LIN {X 0,Y 305.459,Z 160.438,A -85,B 0,C 180,E1 -15804.888,E2 -15804.888} C_VEL
LIN {X 0,Y 305.449,Z 160.435,A -85,B 0,C 180,E1 -15808.356,E2 -15808.356} C_VEL
LIN {X 0,Y 305.518,Z 160.428,A -85,B 0,C 180,E1 -15811.115,E2 -15811.115} C_VEL
LIN {X 0,Y 305.57,Z 160.425,A -85,B 0,C 180,E1 -15814.089,E2 -15814.089} C_VEL
LIN {X 0,Y 305.497,Z 160.431,A -85,B 0,C 180,E1 -15818.404,E2 -15818.404} C_VEL
LIN {X 0,Y 305.556,Z 160.425,A -85,B 0,C 180,E1 -15821.217,E2 -15821.217} C_VEL
LIN {X 0,Y 305.626,Z 160.413,A -85,B 0,C 180,E1 -15825.349,E2 -15825.349} C_VEL
LIN {X 0,Y 305.625,Z 160.413,A -85,B 0,C 180,E1 -15829.4,E2 -15829.4} C_VEL
LIN {X 0,Y 305.749,Z 160.391,A -85,B 0,C 180,E1 -15832.074,E2 -15832.074} C_VEL
LIN {X 0,Y 305.671,Z 160.401,A -85,B 0,C 180,E1 -15834.724,E2 -15834.724} C_VEL
LIN {X 0,Y 305.952,Z 160.37,A -85,B 0,C 180,E1 -15838.685,E2 -15838.685} C_VEL
LIN {X 0,Y 305.948,Z 160.361,A -85,B 0,C 180,E1 -15841.317,E2 -15841.317} C_VEL
LIN {X 0,Y 305.789,Z 160.382,A -85,B 0,C 180,E1 -15846.6,E2 -15846.6} C_VEL
LIN {X 0,Y 305.696,Z 160.401,A -85,B 0,C 180,E1 -15849.262,E2 -15849.262} C_VEL
LIN {X 0,Y 305.587,Z 160.417,A -85,B 0,C 180,E1 -15853.297,E2 -15853.297} C_VEL
LIN {X 0,Y 305.541,Z 160.413,A -85,B 0,C 180,E1 -15856.024,E2 -15856.024} C_VEL
LIN {X 0,Y 305.482,Z 160.427,A -85,B 0,C 180,E1 -15860.189,E2 -15860.189} C_VEL
LIN {X 0,Y 305.442,Z 160.436,A -85,B 0,C 180,E1 -15864.468,E2 -15864.468} C_VEL
LIN {X 0,Y 305.451,Z 160.431,A -85,B 0,C 180,E1 -15867.399,E2 -15867.399} C_VEL
LIN {X 0,Y 305.431,Z 160.429,A -85,B 0,C 180,E1 -15870.414,E2 -15870.414} C_VEL
LIN {X 0,Y 305.467,Z 160.428,A -85,B 0,C 180,E1 -15874.079,E2 -15874.079} C_VEL
LIN {X 0,Y 305.453,Z 160.438,A -85,B 0,C 180,E1 -15876.744,E2 -15876.744} C_VEL
LIN {X 0,Y 305.411,Z 160.442,A -85,B 0,C 180,E1 -15880.59,E2 -15880.59} C_VEL
LIN {X 0,Y 305.423,Z 160.441,A -85,B 0,C 180,E1 -15883.657,E2 -15883.657} C_VEL
LIN {X 0,Y 305.437,Z 160.444,A -85,B 0,C 180,E1 -15887.419,E2 -15887.419} C_VEL
LIN {X 0,Y 305.444,Z 160.439,A -85,B 0,C 180,E1 -15891.593,E2 -15891.593} C_VEL
LIN {X 0,Y 305.489,Z 160.556,A -85,B 0,C 180,E1 -15895.319,E2 -15895.319} C_VEL
LIN {X 0,Y 308.003,Z 170.762,A -85,B 0,C 180,E1 -15898.728,E2 -15898.728} C_VEL
LIN {X 0,Y 309.903,Z 179.796,A -85,B 0,C 180,E1 -15901.56,E2 -15901.56} C_VEL
LIN {X 0,Y 310.831,Z 184.661,A -85,B 0,C 180,E1 -15902.985,E2 -15902.985} C_VEL
LIN {X 0,Y 312.383,Z 189.96,A -85,B 0,C 180,E1 -15903.288,E2 -15903.288} C_VEL
LIN {X 0,Y 316.289,Z 210.278,A -85,B 0,C 180,E1 -15904.21,E2 -15904.21} C_VEL
LIN {X 0,Y 318.973,Z 229.13,A -85,B 0,C 180,E1 -15904.953,E2 -15904.953} C_VEL
LIN {X 0,Y 317.191,Z 294.073,A -85,B 0,C 180,E1 -15906.495,E2 -15906.495} C_VEL
LIN {X 0,Y 316.159,Z 307.688,A -85,B 0,C 180,E1 -15907.064,E2 -15907.064} C_VEL
LIN {X 0,Y 314.832,Z 320.533,A -85,B 0,C 180,E1 -15907.871,E2 -15907.871} C_VEL
LIN {X 0,Y 313.273,Z 333.066,A -85,B 0,C 180,E1 -15908.965,E2 -15908.965} C_VEL
LIN {X 0,Y 311.564,Z 344.273,A -85,B 0,C 180,E1 -15910.223,E2 -15910.223} C_VEL
LIN {X 0,Y 309.857,Z 354.387,A -85,B 0,C 180,E1 -15911.657,E2 -15911.657} C_VEL
LIN {X 0,Y 308.403,Z 363.848,A -85,B 0,C 180,E1 -15913.345,E2 -15913.345} C_VEL
LIN {X 0,Y 307.067,Z 371.791,A -85,B 0,C 180,E1 -15915.079,E2 -15915.079} C_VEL
LIN {X 0,Y 305.664,Z 379.121,A -85,B 0,C 180,E1 -15917.046,E2 -15917.046} C_VEL
LIN {X 0,Y 304.863,Z 384.095,A -85,B 0,C 180,E1 -15918.7,E2 -15918.7} C_VEL
LIN {X 0,Y 304.229,Z 388.944,A -85,B 0,C 180,E1 -15920.694,E2 -15920.694} C_VEL
LIN {X 0,Y 303.828,Z 392.677,A -85,B 0,C 180,E1 -15922.691,E2 -15922.691} C_VEL
LIN {X 0,Y 303.621,Z 395.397,A -85,B 0,C 180,E1 -15924.688,E2 -15924.688} C_VEL
LIN {X 0,Y 303.629,Z 396.691,A -85,B 0,C 180,E1 -15926.018,E2 -15926.018} C_VEL
LIN {X 0,Y 303.624,Z 397.581,A -85,B 0,C 180,E1 -15927.347,E2 -15927.347} C_VEL
LIN {X 0,Y 303.615,Z 398.031,A -85,B 0,C 180,E1 -15928.674,E2 -15928.674} C_VEL
LIN {X 0,Y 303.67,Z 398.088,A -85,B 0,C 180,E1 -15930,E2 -15930} C_VEL
LIN {X 0,Y 303.626,Z 397.751,A -85,B 0,C 180,E1 -15931.327,E2 -15931.327} C_VEL
LIN {X 0,Y 303.626,Z 397.019,A -85,B 0,C 180,E1 -15932.654,E2 -15932.654} C_VEL
LIN {X 0,Y 303.63,Z 395.835,A -85,B 0,C 180,E1 -15933.982,E2 -15933.982} C_VEL
LIN {X 0,Y 303.622,Z 393.936,A -85,B 0,C 180,E1 -15935.532,E2 -15935.532} C_VEL
LIN {X 0,Y 303.927,Z 389.712,A -85,B 0,C 180,E1 -15937.975,E2 -15937.975} C_VEL
LIN {X 0,Y 304.361,Z 385.011,A -85,B 0,C 180,E1 -15939.973,E2 -15939.973} C_VEL
LIN {X 0,Y 305.191,Z 377.914,A -85,B 0,C 180,E1 -15942.299,E2 -15942.299} C_VEL
LIN {X 0,Y 306.358,Z 370.227,A -85,B 0,C 180,E1 -15944.277,E2 -15944.277} C_VEL
LIN {X 0,Y 307.697,Z 360.747,A -85,B 0,C 180,E1 -15946.21,E2 -15946.21} C_VEL
LIN {X 0,Y 309.019,Z 350.537,A -85,B 0,C 180,E1 -15947.881,E2 -15947.881} C_VEL
LIN {X 0,Y 310.561,Z 339.27,A -85,B 0,C 180,E1 -15949.328,E2 -15949.328} C_VEL
LIN {X 0,Y 311.897,Z 328.23,A -85,B 0,C 180,E1 -15950.443,E2 -15950.443} C_VEL
LIN {X 0,Y 313.162,Z 316.02,A -85,B 0,C 180,E1 -15951.389,E2 -15951.389} C_VEL
LIN {X 0,Y 314.23,Z 303.288,A -85,B 0,C 180,E1 -15952.088,E2 -15952.088} C_VEL
LIN {X 0,Y 314.859,Z 290.01,A -85,B 0,C 180,E1 -15952.558,E2 -15952.558} C_VEL
LIN {X 0,Y 316.214,Z 227.211,A -85,B 0,C 180,E1 -15954.02,E2 -15954.02} C_VEL
LIN {X 0,Y 310.529,Z 189.601,A -85,B 0,C 180,E1 -15955.391,E2 -15955.391} C_VEL
LIN {X 0,Y 309.869,Z 185.486,A -85,B 0,C 180,E1 -15955.572,E2 -15955.572} C_VEL
LIN {X 0,Y 309.869,Z 181.695,A -85,B 0,C 180,E1 -15956.612,E2 -15956.612} C_VEL
LIN {X 0,Y 307.783,Z 170.867,A -85,B 0,C 180,E1 -15959.806,E2 -15959.806} C_VEL
LIN {X 0,Y 305.485,Z 160.432,A -85,B 0,C 180,E1 -15963.071,E2 -15963.071} C_VEL
LIN {X 0,Y 305.457,Z 160.435,A -85,B 0,C 180,E1 -15966.743,E2 -15966.743} C_VEL
LIN {X 0,Y 305.414,Z 160.44,A -85,B 0,C 180,E1 -15970.59,E2 -15970.59} C_VEL
LIN {X 0,Y 305.425,Z 160.44,A -85,B 0,C 180,E1 -15973.656,E2 -15973.656} C_VEL
LIN {X 0,Y 305.44,Z 160.44,A -85,B 0,C 180,E1 -15977.418,E2 -15977.418} C_VEL
LIN {X 0,Y 305.465,Z 160.435,A -85,B 0,C 180,E1 -15981.595,E2 -15981.595} C_VEL
LIN {X 0,Y 305.466,Z 160.437,A -85,B 0,C 180,E1 -15984.886,E2 -15984.886} C_VEL
LIN {X 0,Y 305.447,Z 160.436,A -85,B 0,C 180,E1 -15988.358,E2 -15988.358} C_VEL
LIN {X 0,Y 305.48,Z 160.434,A -85,B 0,C 180,E1 -15991.109,E2 -15991.109} C_VEL
LIN {X 0,Y 305.505,Z 160.428,A -85,B 0,C 180,E1 -15994.081,E2 -15994.081} C_VEL
LIN {X 0,Y 305.478,Z 160.434,A -85,B 0,C 180,E1 -15996.975,E2 -15996.975} C_VEL
LIN {X 0,Y 305.513,Z 160.427,A -85,B 0,C 180,E1 -16001.212,E2 -16001.212} C_VEL
LIN {X 0,Y 305.584,Z 160.418,A -85,B 0,C 180,E1 -16005.345,E2 -16005.345} C_VEL
LIN {X 0,Y 305.628,Z 160.41,A -85,B 0,C 180,E1 -16009.398,E2 -16009.398} C_VEL
LIN {X 0,Y 305.751,Z 160.393,A -85,B 0,C 180,E1 -16012.072,E2 -16012.072} C_VEL
LIN {X 0,Y 305.662,Z 160.409,A -85,B 0,C 180,E1 -16014.722,E2 -16014.722} C_VEL
LIN {X 0,Y 305.939,Z 160.374,A -85,B 0,C 180,E1 -16018.683,E2 -16018.683} C_VEL
LIN {X 0,Y 305.939,Z 160.37,A -85,B 0,C 180,E1 -16021.315,E2 -16021.315} C_VEL
LIN {X 0,Y 305.787,Z 160.392,A -85,B 0,C 180,E1 -16026.598,E2 -16026.598} C_VEL
LIN {X 0,Y 305.696,Z 160.404,A -85,B 0,C 180,E1 -16029.26,E2 -16029.26} C_VEL
LIN {X 0,Y 305.572,Z 160.417,A -85,B 0,C 180,E1 -16033.296,E2 -16033.296} C_VEL
LIN {X 0,Y 305.512,Z 160.423,A -85,B 0,C 180,E1 -16036.023,E2 -16036.023} C_VEL
LIN {X 0,Y 305.476,Z 160.432,A -85,B 0,C 180,E1 -16040.187,E2 -16040.187} C_VEL
LIN {X 0,Y 305.439,Z 160.433,A -85,B 0,C 180,E1 -16044.466,E2 -16044.466} C_VEL
LIN {X 0,Y 305.441,Z 160.432,A -85,B 0,C 180,E1 -16047.398,E2 -16047.398} C_VEL
LIN {X 0,Y 305.416,Z 160.437,A -85,B 0,C 180,E1 -16050.413,E2 -16050.413} C_VEL
LIN {X 0,Y 305.463,Z 160.433,A -85,B 0,C 180,E1 -16054.077,E2 -16054.077} C_VEL
LIN {X 0,Y 305.45,Z 160.432,A -85,B 0,C 180,E1 -16056.741,E2 -16056.741} C_VEL
LIN {X 0,Y 305.406,Z 160.438,A -85,B 0,C 180,E1 -16060.588,E2 -16060.588} C_VEL
LIN {X 0,Y 305.417,Z 160.44,A -85,B 0,C 180,E1 -16063.655,E2 -16063.655} C_VEL
LIN {X 0,Y 305.431,Z 160.436,A -85,B 0,C 180,E1 -16067.417,E2 -16067.417} C_VEL
LIN {X 0,Y 305.455,Z 160.435,A -85,B 0,C 180,E1 -16071.594,E2 -16071.594} C_VEL
LIN {X 0,Y 305.456,Z 160.435,A -85,B 0,C 180,E1 -16074.885,E2 -16074.885} C_VEL
LIN {X 0,Y 305.436,Z 160.438,A -85,B 0,C 180,E1 -16078.357,E2 -16078.357} C_VEL
LIN {X 0,Y 305.468,Z 160.432,A -85,B 0,C 180,E1 -16081.108,E2 -16081.108} C_VEL
LIN {X 0,Y 305.472,Z 160.432,A -85,B 0,C 180,E1 -16084.078,E2 -16084.078} C_VEL
LIN {X 0,Y 305.452,Z 160.436,A -85,B 0,C 180,E1 -16088.399,E2 -16088.399} C_VEL
LIN {X 0,Y 305.502,Z 160.429,A -85,B 0,C 180,E1 -16091.212,E2 -16091.212} C_VEL
LIN {X 0,Y 305.572,Z 160.418,A -85,B 0,C 180,E1 -16095.345,E2 -16095.345} C_VEL
LIN {X 0,Y 305.615,Z 160.413,A -85,B 0,C 180,E1 -16099.399,E2 -16099.399} C_VEL
LIN {X 0,Y 305.739,Z 160.401,A -85,B 0,C 180,E1 -16102.072,E2 -16102.072} C_VEL
LIN {X 0,Y 305.65,Z 160.457,A -85,B 0,C 180,E1 -16104.722,E2 -16104.722} C_VEL
LIN {X 0,Y 306.613,Z 165.016,A -85,B 0,C 180,E1 -16106.248,E2 -16106.248} C_VEL
LIN {X 0,Y 312.464,Z 179.943,A -85,B 0,C 180,E1 -16107.106,E2 -16107.106} C_VEL
LIN {X 0,Y 315.894,Z 190.278,A -85,B 0,C 180,E1 -16107.63,E2 -16107.63} C_VEL
LIN {X 0,Y 316.999,Z 196.484,A -85,B 0,C 180,E1 -16107.866,E2 -16107.866} C_VEL
LIN {X 0,Y 314.976,Z 272.651,A -85,B 0,C 180,E1 -16109.64,E2 -16109.64} C_VEL
LIN {X 0,Y 314.278,Z 285.795,A -85,B 0,C 180,E1 -16110.2,E2 -16110.2} C_VEL
LIN {X 0,Y 313.454,Z 297.884,A -85,B 0,C 180,E1 -16110.963,E2 -16110.963} C_VEL
LIN {X 0,Y 312.447,Z 309.33,A -85,B 0,C 180,E1 -16111.933,E2 -16111.933} C_VEL
LIN {X 0,Y 311.048,Z 321.197,A -85,B 0,C 180,E1 -16113.238,E2 -16113.238} C_VEL
LIN {X 0,Y 309.738,Z 331.319,A -85,B 0,C 180,E1 -16114.641,E2 -16114.641} C_VEL
LIN {X 0,Y 308.483,Z 340.503,A -85,B 0,C 180,E1 -16116.212,E2 -16116.212} C_VEL
LIN {X 0,Y 307.288,Z 348.479,A -85,B 0,C 180,E1 -16117.887,E2 -16117.887} C_VEL
LIN {X 0,Y 306.119,Z 356.027,A -85,B 0,C 180,E1 -16119.848,E2 -16119.848} C_VEL
LIN {X 0,Y 305.158,Z 362.491,A -85,B 0,C 180,E1 -16121.963,E2 -16121.963} C_VEL
LIN {X 0,Y 304.444,Z 367.731,A -85,B 0,C 180,E1 -16124.179,E2 -16124.179} C_VEL
LIN {X 0,Y 304.015,Z 371.135,A -85,B 0,C 180,E1 -16126.105,E2 -16126.105} C_VEL
LIN {X 0,Y 303.636,Z 373.968,A -85,B 0,C 180,E1 -16128.383,E2 -16128.383} C_VEL
LIN {X 0,Y 303.447,Z 375.408,A -85,B 0,C 180,E1 -16130.329,E2 -16130.329} C_VEL
LIN {X 0,Y 303.451,Z 375.955,A -85,B 0,C 180,E1 -16132.122,E2 -16132.122} C_VEL
LIN {X 0,Y 303.575,Z 375.564,A -85,B 0,C 180,E1 -16134.627,E2 -16134.627} C_VEL
LIN {X 0,Y 303.751,Z 374.658,A -85,B 0,C 180,E1 -16136.079,E2 -16136.079} C_VEL
LIN {X 0,Y 304.286,Z 371.901,A -85,B 0,C 180,E1 -16138.64,E2 -16138.64} C_VEL
LIN {X 0,Y 304.946,Z 367.905,A -85,B 0,C 180,E1 -16141.021,E2 -16141.021} C_VEL
LIN {X 0,Y 305.631,Z 364.099,A -85,B 0,C 180,E1 -16142.71,E2 -16142.71} C_VEL
LIN {X 0,Y 306.836,Z 357.731,A -85,B 0,C 180,E1 -16144.933,E2 -16144.933} C_VEL
LIN {X 0,Y 308.34,Z 349.761,A -85,B 0,C 180,E1 -16147.086,E2 -16147.086} C_VEL
LIN {X 0,Y 309.942,Z 340.851,A -85,B 0,C 180,E1 -16148.994,E2 -16148.994} C_VEL
LIN {X 0,Y 311.578,Z 331.082,A -85,B 0,C 180,E1 -16150.653,E2 -16150.653} C_VEL
LIN {X 0,Y 313.215,Z 320.303,A -85,B 0,C 180,E1 -16152.118,E2 -16152.118} C_VEL
LIN {X 0,Y 314.771,Z 308.639,A -85,B 0,C 180,E1 -16153.359,E2 -16153.359} C_VEL
LIN {X 0,Y 315.985,Z 296.732,A -85,B 0,C 180,E1 -16154.333,E2 -16154.333} C_VEL
LIN {X 0,Y 316.947,Z 284.09,A -85,B 0,C 180,E1 -16155.093,E2 -16155.093} C_VEL
LIN {X 0,Y 317.614,Z 271.593,A -85,B 0,C 180,E1 -16155.586,E2 -16155.586} C_VEL
LIN {X 0,Y 319.739,Z 196.647,A -85,B 0,C 180,E1 -16157.338,E2 -16157.338} C_VEL
LIN {X 0,Y 318.932,Z 193.583,A -85,B 0,C 180,E1 -16157.495,E2 -16157.495} C_VEL
LIN {X 0,Y 316.079,Z 188.881,A -85,B 0,C 180,E1 -16157.897,E2 -16157.897} C_VEL
LIN {X 0,Y 304.505,Z 175.175,A -85,B 0,C 180,E1 -16159.481,E2 -16159.481} C_VEL
LIN {X 0,Y 301.74,Z 170.475,A -85,B 0,C 180,E1 -16159.924,E2 -16159.924} C_VEL
LIN {X 0,Y 299.63,Z 166.062,A -85,B 0,C 180,E1 -16160.327,E2 -16160.327} C_VEL
LIN {X 0,Y 298.456,Z 161.318,A -85,B 0,C 180,E1 -16162.152,E2 -16162.152} C_VEL
LIN {X 0,Y 298.405,Z 161.318,A -85,B 0,C 180,E1 -16165.582,E2 -16165.582} C_VEL
LIN {X 0,Y 298.392,Z 161.315,A -85,B 0,C 180,E1 -16168.792,E2 -16168.792} C_VEL
LIN {X 0,Y 298.461,Z 161.309,A -85,B 0,C 180,E1 -16171.906,E2 -16171.906} C_VEL
LIN {X 0,Y 298.484,Z 161.307,A -85,B 0,C 180,E1 -16174.925,E2 -16174.925} C_VEL
LIN {X 0,Y 298.444,Z 161.306,A -85,B 0,C 180,E1 -16179.316,E2 -16179.316} C_VEL
LIN {X 0,Y 298.508,Z 161.298,A -85,B 0,C 180,E1 -16182.179,E2 -16182.179} C_VEL
LIN {X 0,Y 298.585,Z 161.293,A -85,B 0,C 180,E1 -16184.996,E2 -16184.996} C_VEL
LIN {X 0,Y 298.583,Z 161.292,A -85,B 0,C 180,E1 -16189.147,E2 -16189.147} C_VEL
LIN {X 0,Y 298.7,Z 161.269,A -85,B 0,C 180,E1 -16191.886,E2 -16191.886} C_VEL
LIN {X 0,Y 298.639,Z 161.278,A -85,B 0,C 180,E1 -16194.6,E2 -16194.6} C_VEL
LIN {X 0,Y 298.919,Z 161.246,A -85,B 0,C 180,E1 -16198.654,E2 -16198.654} C_VEL
LIN {X 0,Y 298.915,Z 161.236,A -85,B 0,C 180,E1 -16201.348,E2 -16201.348} C_VEL
LIN {X 0,Y 298.737,Z 161.261,A -85,B 0,C 180,E1 -16206.756,E2 -16206.756} C_VEL
LIN {X 0,Y 298.628,Z 161.283,A -85,B 0,C 180,E1 -16209.483,E2 -16209.483} C_VEL
LIN {X 0,Y 298.543,Z 161.297,A -85,B 0,C 180,E1 -16213.617,E2 -16213.617} C_VEL
LIN {X 0,Y 298.473,Z 161.293,A -85,B 0,C 180,E1 -16216.414,E2 -16216.414} C_VEL
LIN {X 0,Y 298.441,Z 161.31,A -85,B 0,C 180,E1 -16219.616,E2 -16219.616} C_VEL
LIN {X 0,Y 298.384,Z 161.317,A -85,B 0,C 180,E1 -16223.605,E2 -16223.605} C_VEL
LIN {X 0,Y 298.404,Z 161.304,A -85,B 0,C 180,E1 -16226.584,E2 -16226.584} C_VEL
LIN {X 0,Y 298.395,Z 161.309,A -85,B 0,C 180,E1 -16229.645,E2 -16229.645} C_VEL
LIN {X 0,Y 298.395,Z 161.316,A -85,B 0,C 180,E1 -16232.801,E2 -16232.801} C_VEL
LIN {X 0,Y 298.428,Z 161.313,A -85,B 0,C 180,E1 -16236.803,E2 -16236.803} C_VEL
LIN {X 0,Y 298.349,Z 161.32,A -85,B 0,C 180,E1 -16241.269,E2 -16241.269} C_VEL
LIN {X 0,Y 298.357,Z 161.326,A -85,B 0,C 180,E1 -16245.036,E2 -16245.036} C_VEL
LIN {X 0,Y 298.35,Z 161.324,A -85,B 0,C 180,E1 -16248.922,E2 -16248.922} C_VEL
LIN {X 0,Y 298.429,Z 161.303,A -85,B 0,C 180,E1 -16253.198,E2 -16253.198} C_VEL
LIN {X 0,Y 298.463,Z 161.48,A -85,B 0,C 180,E1 -16254.662,E2 -16254.662} C_VEL
LIN {X 0,Y 301.06,Z 172.051,A -85,B 0,C 180,E1 -16258.315,E2 -16258.315} C_VEL
LIN {X 0,Y 303.12,Z 181.821,A -85,B 0,C 180,E1 -16261.46,E2 -16261.46} C_VEL
LIN {X 0,Y 303.597,Z 184.363,A -85,B 0,C 180,E1 -16262.2,E2 -16262.2} C_VEL
LIN {X 0,Y 306.198,Z 191.246,A -85,B 0,C 180,E1 -16262.674,E2 -16262.674} C_VEL
LIN {X 0,Y 309.548,Z 208.929,A -85,B 0,C 180,E1 -16263.508,E2 -16263.508} C_VEL
LIN {X 0,Y 312.601,Z 228.987,A -85,B 0,C 180,E1 -16264.345,E2 -16264.345} C_VEL
LIN {X 0,Y 310.814,Z 293.869,A -85,B 0,C 180,E1 -16265.925,E2 -16265.925} C_VEL
LIN {X 0,Y 309.741,Z 307.694,A -85,B 0,C 180,E1 -16266.516,E2 -16266.516} C_VEL
LIN {X 0,Y 308.434,Z 319.935,A -85,B 0,C 180,E1 -16267.298,E2 -16267.298} C_VEL
LIN {X 0,Y 306.894,Z 331.737,A -85,B 0,C 180,E1 -16268.33,E2 -16268.33} C_VEL
LIN {X 0,Y 305.11,Z 343.124,A -85,B 0,C 180,E1 -16269.611,E2 -16269.611} C_VEL
LIN {X 0,Y 303.315,Z 353.421,A -85,B 0,C 180,E1 -16271.072,E2 -16271.072} C_VEL
LIN {X 0,Y 301.751,Z 362.726,A -85,B 0,C 180,E1 -16272.733,E2 -16272.733} C_VEL
LIN {X 0,Y 300.168,Z 371.722,A -85,B 0,C 180,E1 -16274.728,E2 -16274.728} C_VEL
LIN {X 0,Y 298.739,Z 379.02,A -85,B 0,C 180,E1 -16276.74,E2 -16276.74} C_VEL
LIN {X 0,Y 297.864,Z 383.964,A -85,B 0,C 180,E1 -16278.431,E2 -16278.431} C_VEL
LIN {X 0,Y 297.202,Z 388.786,A -85,B 0,C 180,E1 -16280.472,E2 -16280.472} C_VEL
LIN {X 0,Y 296.777,Z 392.494,A -85,B 0,C 180,E1 -16282.516,E2 -16282.516} C_VEL
LIN {X 0,Y 296.535,Z 395.188,A -85,B 0,C 180,E1 -16284.56,E2 -16284.56} C_VEL
LIN {X 0,Y 296.526,Z 396.472,A -85,B 0,C 180,E1 -16285.923,E2 -16285.923} C_VEL
LIN {X 0,Y 296.549,Z 397.343,A -85,B 0,C 180,E1 -16287.284,E2 -16287.284} C_VEL
LIN {X 0,Y 296.532,Z 397.776,A -85,B 0,C 180,E1 -16288.642,E2 -16288.642} C_VEL
LIN {X 0,Y 296.582,Z 397.822,A -85,B 0,C 180,E1 -16290,E2 -16290} C_VEL
LIN {X 0,Y 296.542,Z 397.474,A -85,B 0,C 180,E1 -16291.358,E2 -16291.358} C_VEL
LIN {X 0,Y 296.551,Z 396.723,A -85,B 0,C 180,E1 -16292.717,E2 -16292.717} C_VEL
LIN {X 0,Y 296.526,Z 395.521,A -85,B 0,C 180,E1 -16294.078,E2 -16294.078} C_VEL
LIN {X 0,Y 296.55,Z 393.815,A -85,B 0,C 180,E1 -16295.509,E2 -16295.509} C_VEL
LIN {X 0,Y 296.777,Z 390.651,A -85,B 0,C 180,E1 -16297.484,E2 -16297.484} C_VEL
LIN {X 0,Y 297.144,Z 386.308,A -85,B 0,C 180,E1 -16299.53,E2 -16299.53} C_VEL
LIN {X 0,Y 297.751,Z 380.757,A -85,B 0,C 180,E1 -16301.574,E2 -16301.574} C_VEL
LIN {X 0,Y 298.817,Z 373.827,A -85,B 0,C 180,E1 -16303.603,E2 -16303.603} C_VEL
LIN {X 0,Y 299.877,Z 366.738,A -85,B 0,C 180,E1 -16305.288,E2 -16305.288} C_VEL
LIN {X 0,Y 301.068,Z 358.157,A -85,B 0,C 180,E1 -16306.969,E2 -16306.969} C_VEL
LIN {X 0,Y 302.376,Z 348.77,A -85,B 0,C 180,E1 -16308.463,E2 -16308.463} C_VEL
LIN {X 0,Y 304.007,Z 337.12,A -85,B 0,C 180,E1 -16309.938,E2 -16309.938} C_VEL
LIN {X 0,Y 305.466,Z 325.624,A -85,B 0,C 180,E1 -16311.069,E2 -16311.069} C_VEL
LIN {X 0,Y 306.713,Z 313.738,A -85,B 0,C 180,E1 -16311.95,E2 -16311.95} C_VEL
LIN {X 0,Y 307.71,Z 300.045,A -85,B 0,C 180,E1 -16312.67,E2 -16312.67} C_VEL
LIN {X 0,Y 308.277,Z 287.167,A -85,B 0,C 180,E1 -16313.085,E2 -16313.085} C_VEL
LIN {X 0,Y 309.61,Z 227.825,A -85,B 0,C 180,E1 -16314.488,E2 -16314.488} C_VEL
LIN {X 0,Y 304.096,Z 191.169,A -85,B 0,C 180,E1 -16315.864,E2 -16315.864} C_VEL
LIN {X 0,Y 303.048,Z 185.178,A -85,B 0,C 180,E1 -16316.144,E2 -16316.144} C_VEL
LIN {X 0,Y 302.253,Z 179.1,A -85,B 0,C 180,E1 -16317.921,E2 -16317.921} C_VEL
LIN {X 0,Y 299.648,Z 166.678,A -85,B 0,C 180,E1 -16321.76,E2 -16321.76} C_VEL
LIN {X 0,Y 298.438,Z 161.309,A -85,B 0,C 180,E1 -16323.501,E2 -16323.501} C_VEL
LIN {X 0,Y 298.395,Z 161.315,A -85,B 0,C 180,E1 -16327.762,E2 -16327.762} C_VEL
LIN {X 0,Y 298.352,Z 161.322,A -85,B 0,C 180,E1 -16331.268,E2 -16331.268} C_VEL
LIN {X 0,Y 298.359,Z 161.321,A -85,B 0,C 180,E1 -16335.035,E2 -16335.035} C_VEL
LIN {X 0,Y 298.353,Z 161.322,A -85,B 0,C 180,E1 -16338.921,E2 -16338.921} C_VEL
LIN {X 0,Y 298.446,Z 161.312,A -85,B 0,C 180,E1 -16343.194,E2 -16343.194} C_VEL
LIN {X 0,Y 298.398,Z 161.317,A -85,B 0,C 180,E1 -16347.199,E2 -16347.199} C_VEL
LIN {X 0,Y 298.407,Z 161.315,A -85,B 0,C 180,E1 -16350.624,E2 -16350.624} C_VEL
LIN {X 0,Y 298.444,Z 161.312,A -85,B 0,C 180,E1 -16354.919,E2 -16354.919} C_VEL
LIN {X 0,Y 298.403,Z 161.312,A -85,B 0,C 180,E1 -16357.861,E2 -16357.861} C_VEL
LIN {X 0,Y 298.464,Z 161.309,A -85,B 0,C 180,E1 -16360.751,E2 -16360.751} C_VEL
LIN {X 0,Y 298.515,Z 161.3,A -85,B 0,C 180,E1 -16364.99,E2 -16364.99} C_VEL
LIN {X 0,Y 298.587,Z 161.287,A -85,B 0,C 180,E1 -16369.145,E2 -16369.145} C_VEL
LIN {X 0,Y 298.702,Z 161.269,A -85,B 0,C 180,E1 -16371.883,E2 -16371.883} C_VEL
LIN {X 0,Y 298.632,Z 161.285,A -85,B 0,C 180,E1 -16374.597,E2 -16374.597} C_VEL
LIN {X 0,Y 298.907,Z 161.25,A -85,B 0,C 180,E1 -16378.652,E2 -16378.652} C_VEL
LIN {X 0,Y 298.907,Z 161.246,A -85,B 0,C 180,E1 -16381.346,E2 -16381.346} C_VEL
LIN {X 0,Y 298.736,Z 161.269,A -85,B 0,C 180,E1 -16386.754,E2 -16386.754} C_VEL
LIN {X 0,Y 298.628,Z 161.285,A -85,B 0,C 180,E1 -16389.481,E2 -16389.481} C_VEL
LIN {X 0,Y 298.524,Z 161.297,A -85,B 0,C 180,E1 -16393.615,E2 -16393.615} C_VEL
LIN {X 0,Y 298.452,Z 161.3,A -85,B 0,C 180,E1 -16396.413,E2 -16396.413} C_VEL
LIN {X 0,Y 298.432,Z 161.31,A -85,B 0,C 180,E1 -16399.61,E2 -16399.61} C_VEL
LIN {X 0,Y 298.382,Z 161.318,A -85,B 0,C 180,E1 -16403.603,E2 -16403.603} C_VEL
LIN {X 0,Y 298.4,Z 161.305,A -85,B 0,C 180,E1 -16406.582,E2 -16406.582} C_VEL
LIN {X 0,Y 298.356,Z 161.319,A -85,B 0,C 180,E1 -16409.647,E2 -16409.647} C_VEL
LIN {X 0,Y 298.392,Z 161.314,A -85,B 0,C 180,E1 -16412.799,E2 -16412.799} C_VEL
LIN {X 0,Y 298.424,Z 161.307,A -85,B 0,C 180,E1 -16416.801,E2 -16416.801} C_VEL
LIN {X 0,Y 298.345,Z 161.321,A -85,B 0,C 180,E1 -16421.078,E2 -16421.078} C_VEL
LIN {X 0,Y 298.351,Z 161.322,A -85,B 0,C 180,E1 -16425.034,E2 -16425.034} C_VEL
LIN {X 0,Y 298.344,Z 161.32,A -85,B 0,C 180,E1 -16428.92,E2 -16428.92} C_VEL
LIN {X 0,Y 298.393,Z 161.315,A -85,B 0,C 180,E1 -16432.238,E2 -16432.238} C_VEL
LIN {X 0,Y 298.403,Z 161.311,A -85,B 0,C 180,E1 -16435.58,E2 -16435.58} C_VEL
LIN {X 0,Y 298.372,Z 161.321,A -85,B 0,C 180,E1 -16438.788,E2 -16438.788} C_VEL
LIN {X 0,Y 298.403,Z 161.31,A -85,B 0,C 180,E1 -16441.898,E2 -16441.898} C_VEL
LIN {X 0,Y 298.407,Z 161.313,A -85,B 0,C 180,E1 -16444.917,E2 -16444.917} C_VEL
LIN {X 0,Y 298.384,Z 161.313,A -85,B 0,C 180,E1 -16447.86,E2 -16447.86} C_VEL
LIN {X 0,Y 298.453,Z 161.31,A -85,B 0,C 180,E1 -16450.751,E2 -16450.751} C_VEL
LIN {X 0,Y 298.504,Z 161.299,A -85,B 0,C 180,E1 -16454.99,E2 -16454.99} C_VEL
LIN {X 0,Y 298.574,Z 161.291,A -85,B 0,C 180,E1 -16459.146,E2 -16459.146} C_VEL
LIN {X 0,Y 298.691,Z 161.278,A -85,B 0,C 180,E1 -16461.884,E2 -16461.884} C_VEL
LIN {X 0,Y 298.661,Z 161.47,A -85,B 0,C 180,E1 -16464.345,E2 -16464.345} C_VEL
LIN {X 0,Y 299.481,Z 165.574,A -85,B 0,C 180,E1 -16465.668,E2 -16465.668} C_VEL
LIN {X 0,Y 305.39,Z 180.099,A -85,B 0,C 180,E1 -16466.545,E2 -16466.545} C_VEL
LIN {X 0,Y 309.453,Z 191.955,A -85,B 0,C 180,E1 -16467.177,E2 -16467.177} C_VEL
LIN {X 0,Y 310.405,Z 197.984,A -85,B 0,C 180,E1 -16467.404,E2 -16467.404} C_VEL
LIN {X 0,Y 308.344,Z 272.826,A -85,B 0,C 180,E1 -16469.183,E2 -16469.183} C_VEL
LIN {X 0,Y 307.606,Z 286.01,A -85,B 0,C 180,E1 -16469.754,E2 -16469.754} C_VEL
LIN {X 0,Y 306.699,Z 298.681,A -85,B 0,C 180,E1 -16470.574,E2 -16470.574} C_VEL
LIN {X 0,Y 305.559,Z 310.779,A -85,B 0,C 180,E1 -16471.647,E2 -16471.647} C_VEL
LIN {X 0,Y 304.164,Z 322.407,A -85,B 0,C 180,E1 -16472.98,E2 -16472.98} C_VEL
LIN {X 0,Y 302.8,Z 332.396,A -85,B 0,C 180,E1 -16474.417,E2 -16474.417} C_VEL
LIN {X 0,Y 301.494,Z 341.391,A -85,B 0,C 180,E1 -16476.021,E2 -16476.021} C_VEL
LIN {X 0,Y 300.032,Z 350.652,A -85,B 0,C 180,E1 -16478.079,E2 -16478.079} C_VEL
LIN {X 0,Y 298.868,Z 358.091,A -85,B 0,C 180,E1 -16480.158,E2 -16480.158} C_VEL
LIN {X 0,Y 297.949,Z 363.988,A -85,B 0,C 180,E1 -16482.256,E2 -16482.256} C_VEL
LIN {X 0,Y 297.343,Z 368.455,A -85,B 0,C 180,E1 -16484.292,E2 -16484.292} C_VEL
LIN {X 0,Y 296.817,Z 372.082,A -85,B 0,C 180,E1 -16486.507,E2 -16486.507} C_VEL
LIN {X 0,Y 296.526,Z 374.402,A -85,B 0,C 180,E1 -16488.555,E2 -16488.555} C_VEL
LIN {X 0,Y 296.333,Z 375.876,A -85,B 0,C 180,E1 -16490.839,E2 -16490.839} C_VEL
LIN {X 0,Y 296.353,Z 376.24,A -85,B 0,C 180,E1 -16492.353,E2 -16492.353} C_VEL
LIN {X 0,Y 296.397,Z 376.15,A -85,B 0,C 180,E1 -16493.772,E2 -16493.772} C_VEL
LIN {X 0,Y 296.634,Z 375.237,A -85,B 0,C 180,E1 -16495.804,E2 -16495.804} C_VEL
LIN {X 0,Y 297.087,Z 372.953,A -85,B 0,C 180,E1 -16498.237,E2 -16498.237} C_VEL
LIN {X 0,Y 297.689,Z 369.597,A -85,B 0,C 180,E1 -16500.503,E2 -16500.503} C_VEL
LIN {X 0,Y 298.586,Z 364.914,A -85,B 0,C 180,E1 -16502.777,E2 -16502.777} C_VEL
LIN {X 0,Y 299.666,Z 359.388,A -85,B 0,C 180,E1 -16504.833,E2 -16504.833} C_VEL
LIN {X 0,Y 301.103,Z 352.204,A -85,B 0,C 180,E1 -16506.943,E2 -16506.943} C_VEL
LIN {X 0,Y 302.643,Z 344.105,A -85,B 0,C 180,E1 -16508.829,E2 -16508.829} C_VEL
LIN {X 0,Y 304.495,Z 334.068,A -85,B 0,C 180,E1 -16510.695,E2 -16510.695} C_VEL
LIN {X 0,Y 306.116,Z 324.382,A -85,B 0,C 180,E1 -16512.137,E2 -16512.137} C_VEL
LIN {X 0,Y 307.716,Z 313.065,A -85,B 0,C 180,E1 -16513.474,E2 -16513.474} C_VEL
LIN {X 0,Y 309.176,Z 301.04,A -85,B 0,C 180,E1 -16514.574,E2 -16514.574} C_VEL
LIN {X 0,Y 310.282,Z 288.488,A -85,B 0,C 180,E1 -16515.432,E2 -16515.432} C_VEL
LIN {X 0,Y 311.068,Z 275.418,A -85,B 0,C 180,E1 -16516.036,E2 -16516.036} C_VEL
LIN {X 0,Y 311.827,Z 253.176,A -85,B 0,C 180,E1 -16516.615,E2 -16516.615} C_VEL
LIN {X 0,Y 313.503,Z 198.025,A -85,B 0,C 180,E1 -16517.91,E2 -16517.91} C_VEL
LIN {X 0,Y 308.411,Z 184.801,A -85,B 0,C 180,E1 -16518.79,E2 -16518.79} C_VEL
LIN {X 0,Y 301.74,Z 170.475,A -85,B 0,C 180,E1 -16519.924,E2 -16519.924} C_VEL
LIN {X 0,Y 300.083,Z 168.162,A -85,B 0,C 180,E1 -16520.222,E2 -16520.222} C_VEL
LIN {X 0,Y 297.189,Z 166.074,A -85,B 0,C 180,E1 -16520.799,E2 -16520.799} C_VEL
LIN {X 0,Y 294.019,Z 164.514,A -85,B 0,C 180,E1 -16521.613,E2 -16521.613} C_VEL
LIN {X 0,Y 292.194,Z 163.217,A -85,B 0,C 180,E1 -16522.333,E2 -16522.333} C_VEL
LIN {X 0,Y 291.422,Z 162.201,A -85,B 0,C 180,E1 -16523.064,E2 -16523.064} C_VEL
LIN {X 0,Y 291.411,Z 162.19,A -85,B 0,C 180,E1 -16523.134,E2 -16523.134} C_VEL
LIN {X 0,Y 291.342,Z 162.194,A -85,B 0,C 180,E1 -16526.303,E2 -16526.303} C_VEL
LIN {X 0,Y 291.385,Z 162.185,A -85,B 0,C 180,E1 -16530.261,E2 -16530.261} C_VEL
LIN {X 0,Y 291.415,Z 162.188,A -85,B 0,C 180,E1 -16534.273,E2 -16534.273} C_VEL
LIN {X 0,Y 291.38,Z 162.195,A -85,B 0,C 180,E1 -16537.301,E2 -16537.301} C_VEL
LIN {X 0,Y 291.457,Z 162.18,A -85,B 0,C 180,E1 -16540.271,E2 -16540.271} C_VEL
LIN {X 0,Y 291.497,Z 162.176,A -85,B 0,C 180,E1 -16544.666,E2 -16544.666} C_VEL
LIN {X 0,Y 291.529,Z 162.173,A -85,B 0,C 180,E1 -16548.882,E2 -16548.882} C_VEL
LIN {X 0,Y 291.653,Z 162.145,A -85,B 0,C 180,E1 -16551.688,E2 -16551.688} C_VEL
LIN {X 0,Y 291.608,Z 162.155,A -85,B 0,C 180,E1 -16554.469,E2 -16554.469} C_VEL
LIN {X 0,Y 291.885,Z 162.122,A -85,B 0,C 180,E1 -16558.621,E2 -16558.621} C_VEL
LIN {X 0,Y 291.881,Z 162.112,A -85,B 0,C 180,E1 -16561.381,E2 -16561.381} C_VEL
LIN {X 0,Y 291.689,Z 162.141,A -85,B 0,C 180,E1 -16566.92,E2 -16566.92} C_VEL
LIN {X 0,Y 291.57,Z 162.158,A -85,B 0,C 180,E1 -16569.715,E2 -16569.715} C_VEL
LIN {X 0,Y 291.505,Z 162.175,A -85,B 0,C 180,E1 -16573.952,E2 -16573.952} C_VEL
LIN {X 0,Y 291.42,Z 162.172,A -85,B 0,C 180,E1 -16576.823,E2 -16576.823} C_VEL
LIN {X 0,Y 291.393,Z 162.185,A -85,B 0,C 180,E1 -16579.843,E2 -16579.843} C_VEL
LIN {X 0,Y 291.328,Z 162.195,A -85,B 0,C 180,E1 -16584.213,E2 -16584.213} C_VEL
LIN {X 0,Y 291.352,Z 162.186,A -85,B 0,C 180,E1 -16587.28,E2 -16587.28} C_VEL
LIN {X 0,Y 291.32,Z 162.187,A -85,B 0,C 180,E1 -16590.44,E2 -16590.44} C_VEL
LIN {X 0,Y 291.346,Z 162.188,A -85,B 0,C 180,E1 -16593.699,E2 -16593.699} C_VEL
LIN {X 0,Y 291.355,Z 162.189,A -85,B 0,C 180,E1 -16597.249,E2 -16597.249} C_VEL
LIN {X 0,Y 291.296,Z 162.199,A -85,B 0,C 180,E1 -16601.589,E2 -16601.589} C_VEL
LIN {X 0,Y 291.284,Z 162.208,A -85,B 0,C 180,E1 -16605.597,E2 -16605.597} C_VEL
LIN {X 0,Y 291.296,Z 162.203,A -85,B 0,C 180,E1 -16609.351,E2 -16609.351} C_VEL
LIN {X 0,Y 291.371,Z 162.188,A -85,B 0,C 180,E1 -16613.883,E2 -16613.883} C_VEL
LIN {X 0,Y 293.506,Z 170.65,A -85,B 0,C 180,E1 -16616.939,E2 -16616.939} C_VEL
LIN {X 0,Y 295.831,Z 181.007,A -85,B 0,C 180,E1 -16620.441,E2 -16620.441} C_VEL
LIN {X 0,Y 296.424,Z 184.06,A -85,B 0,C 180,E1 -16621.372,E2 -16621.372} C_VEL
LIN {X 0,Y 300.271,Z 193.592,A -85,B 0,C 180,E1 -16622.088,E2 -16622.088} C_VEL
LIN {X 0,Y 303.368,Z 210.21,A -85,B 0,C 180,E1 -16622.895,E2 -16622.895} C_VEL
LIN {X 0,Y 306.302,Z 229.556,A -85,B 0,C 180,E1 -16623.736,E2 -16623.736} C_VEL
LIN {X 0,Y 304.478,Z 293.583,A -85,B 0,C 180,E1 -16625.328,E2 -16625.328} C_VEL
LIN {X 0,Y 303.333,Z 307.701,A -85,B 0,C 180,E1 -16625.944,E2 -16625.944} C_VEL
LIN {X 0,Y 301.926,Z 320.348,A -85,B 0,C 180,E1 -16626.78,E2 -16626.78} C_VEL
LIN {X 0,Y 300.304,Z 332.008,A -85,B 0,C 180,E1 -16627.829,E2 -16627.829} C_VEL
LIN {X 0,Y 298.484,Z 343.297,A -85,B 0,C 180,E1 -16629.138,E2 -16629.138} C_VEL
LIN {X 0,Y 296.621,Z 353.503,A -85,B 0,C 180,E1 -16630.628,E2 -16630.628} C_VEL
LIN {X 0,Y 294.848,Z 363.35,A -85,B 0,C 180,E1 -16632.45,E2 -16632.45} C_VEL
LIN {X 0,Y 293.286,Z 371.681,A -85,B 0,C 180,E1 -16634.361,E2 -16634.361} C_VEL
LIN {X 0,Y 291.824,Z 378.932,A -85,B 0,C 180,E1 -16636.42,E2 -16636.42} C_VEL
LIN {X 0,Y 290.881,Z 383.838,A -85,B 0,C 180,E1 -16638.149,E2 -16638.149} C_VEL
LIN {X 0,Y 290.159,Z 388.627,A -85,B 0,C 180,E1 -16640.239,E2 -16640.239} C_VEL
LIN {X 0,Y 289.708,Z 392.31,A -85,B 0,C 180,E1 -16642.333,E2 -16642.333} C_VEL
LIN {X 0,Y 289.441,Z 395.158,A -85,B 0,C 180,E1 -16644.592,E2 -16644.592} C_VEL
LIN {X 0,Y 289.474,Z 397.101,A -85,B 0,C 180,E1 -16647.217,E2 -16647.217} C_VEL
LIN {X 0,Y 289.451,Z 397.522,A -85,B 0,C 180,E1 -16648.609,E2 -16648.609} C_VEL
LIN {X 0,Y 289.497,Z 397.556,A -85,B 0,C 180,E1 -16650,E2 -16650} C_VEL
LIN {X 0,Y 289.461,Z 397.196,A -85,B 0,C 180,E1 -16651.392,E2 -16651.392} C_VEL
LIN {X 0,Y 289.476,Z 396.424,A -85,B 0,C 180,E1 -16652.783,E2 -16652.783} C_VEL
LIN {X 0,Y 289.435,Z 393.805,A -85,B 0,C 180,E1 -16655.397,E2 -16655.397} C_VEL
LIN {X 0,Y 289.707,Z 390.295,A -85,B 0,C 180,E1 -16657.668,E2 -16657.668} C_VEL
LIN {X 0,Y 290.111,Z 385.922,A -85,B 0,C 180,E1 -16659.764,E2 -16659.764} C_VEL
LIN {X 0,Y 290.758,Z 380.338,A -85,B 0,C 180,E1 -16661.857,E2 -16661.857} C_VEL
LIN {X 0,Y 291.902,Z 373.372,A -85,B 0,C 180,E1 -16663.932,E2 -16663.932} C_VEL
LIN {X 0,Y 293.015,Z 366.242,A -85,B 0,C 180,E1 -16665.655,E2 -16665.655} C_VEL
LIN {X 0,Y 294.235,Z 357.609,A -85,B 0,C 180,E1 -16667.371,E2 -16667.371} C_VEL
LIN {X 0,Y 295.647,Z 348.139,A -85,B 0,C 180,E1 -16668.899,E2 -16668.899} C_VEL
LIN {X 0,Y 297.308,Z 336.405,A -85,B 0,C 180,E1 -16670.406,E2 -16670.406} C_VEL
LIN {X 0,Y 298.84,Z 324.749,A -85,B 0,C 180,E1 -16671.56,E2 -16671.56} C_VEL
LIN {X 0,Y 300.144,Z 312.656,A -85,B 0,C 180,E1 -16672.456,E2 -16672.456} C_VEL
LIN {X 0,Y 301.11,Z 299.541,A -85,B 0,C 180,E1 -16673.15,E2 -16673.15} C_VEL
LIN {X 0,Y 301.728,Z 285.533,A -85,B 0,C 180,E1 -16673.594,E2 -16673.594} C_VEL
LIN {X 0,Y 303.049,Z 228.772,A -85,B 0,C 180,E1 -16674.966,E2 -16674.966} C_VEL
LIN {X 0,Y 297.596,Z 192.452,A -85,B 0,C 180,E1 -16676.367,E2 -16676.367} C_VEL
LIN {X 0,Y 296.077,Z 184.998,A -85,B 0,C 180,E1 -16676.713,E2 -16676.713} C_VEL
LIN {X 0,Y 294.243,Z 175.265,A -85,B 0,C 180,E1 -16679.711,E2 -16679.711} C_VEL
LIN {X 0,Y 292.008,Z 164.919,A -85,B 0,C 180,E1 -16683.047,E2 -16683.047} C_VEL
LIN {X 0,Y 291.399,Z 162.187,A -85,B 0,C 180,E1 -16683.994,E2 -16683.994} C_VEL
LIN {X 0,Y 291.36,Z 162.195,A -85,B 0,C 180,E1 -16687.248,E2 -16687.248} C_VEL
LIN {X 0,Y 291.3,Z 162.197,A -85,B 0,C 180,E1 -16691.588,E2 -16691.588} C_VEL
LIN {X 0,Y 291.287,Z 162.202,A -85,B 0,C 180,E1 -16695.596,E2 -16695.596} C_VEL
LIN {X 0,Y 291.305,Z 162.202,A -85,B 0,C 180,E1 -16699.352,E2 -16699.352} C_VEL
LIN {X 0,Y 291.405,Z 162.189,A -85,B 0,C 180,E1 -16702.918,E2 -16702.918} C_VEL
LIN {X 0,Y 291.349,Z 162.192,A -85,B 0,C 180,E1 -16706.301,E2 -16706.301} C_VEL
LIN {X 0,Y 291.37,Z 162.189,A -85,B 0,C 180,E1 -16710.267,E2 -16710.267} C_VEL
LIN {X 0,Y 291.364,Z 162.19,A -85,B 0,C 180,E1 -16714.266,E2 -16714.266} C_VEL
LIN {X 0,Y 291.367,Z 162.19,A -85,B 0,C 180,E1 -16717.297,E2 -16717.297} C_VEL
LIN {X 0,Y 291.394,Z 162.186,A -85,B 0,C 180,E1 -16720.265,E2 -16720.265} C_VEL
LIN {X 0,Y 291.478,Z 162.179,A -85,B 0,C 180,E1 -16724.682,E2 -16724.682} C_VEL
LIN {X 0,Y 291.532,Z 162.167,A -85,B 0,C 180,E1 -16728.879,E2 -16728.879} C_VEL
LIN {X 0,Y 291.655,Z 162.145,A -85,B 0,C 180,E1 -16731.686,E2 -16731.686} C_VEL
LIN {X 0,Y 291.602,Z 162.16,A -85,B 0,C 180,E1 -16734.467,E2 -16734.467} C_VEL
LIN {X 0,Y 291.874,Z 162.127,A -85,B 0,C 180,E1 -16738.619,E2 -16738.619} C_VEL
LIN {X 0,Y 291.874,Z 162.121,A -85,B 0,C 180,E1 -16741.379,E2 -16741.379} C_VEL
LIN {X 0,Y 291.689,Z 162.147,A -85,B 0,C 180,E1 -16746.918,E2 -16746.918} C_VEL
LIN {X 0,Y 291.57,Z 162.166,A -85,B 0,C 180,E1 -16749.713,E2 -16749.713} C_VEL
LIN {X 0,Y 291.482,Z 162.17,A -85,B 0,C 180,E1 -16753.951,E2 -16753.951} C_VEL
LIN {X 0,Y 291.404,Z 162.176,A -85,B 0,C 180,E1 -16756.822,E2 -16756.822} C_VEL
LIN {X 0,Y 291.392,Z 162.189,A -85,B 0,C 180,E1 -16759.841,E2 -16759.841} C_VEL
LIN {X 0,Y 291.326,Z 162.192,A -85,B 0,C 180,E1 -16764.21,E2 -16764.21} C_VEL
LIN {X 0,Y 291.328,Z 162.187,A -85,B 0,C 180,E1 -16767.28,E2 -16767.28} C_VEL
LIN {X 0,Y 291.301,Z 162.195,A -85,B 0,C 180,E1 -16770.439,E2 -16770.439} C_VEL
LIN {X 0,Y 291.342,Z 162.194,A -85,B 0,C 180,E1 -16773.697,E2 -16773.697} C_VEL
LIN {X 0,Y 291.353,Z 162.187,A -85,B 0,C 180,E1 -16777.247,E2 -16777.247} C_VEL
LIN {X 0,Y 291.296,Z 162.196,A -85,B 0,C 180,E1 -16780.647,E2 -16780.647} C_VEL
LIN {X 0,Y 291.278,Z 162.2,A -85,B 0,C 180,E1 -16784.402,E2 -16784.402} C_VEL
LIN {X 0,Y 291.291,Z 162.195,A -85,B 0,C 180,E1 -16788.41,E2 -16788.41} C_VEL
LIN {X 0,Y 291.33,Z 162.198,A -85,B 0,C 180,E1 -16791.154,E2 -16791.154} C_VEL
LIN {X 0,Y 291.35,Z 162.191,A -85,B 0,C 180,E1 -16794.624,E2 -16794.624} C_VEL
LIN {X 0,Y 291.361,Z 162.19,A -85,B 0,C 180,E1 -16797.949,E2 -16797.949} C_VEL
LIN {X 0,Y 291.336,Z 162.192,A -85,B 0,C 180,E1 -16801.153,E2 -16801.153} C_VEL
LIN {X 0,Y 291.336,Z 162.195,A -85,B 0,C 180,E1 -16804.264,E2 -16804.264} C_VEL
LIN {X 0,Y 291.343,Z 162.19,A -85,B 0,C 180,E1 -16807.296,E2 -16807.296} C_VEL
LIN {X 0,Y 291.378,Z 162.191,A -85,B 0,C 180,E1 -16810.264,E2 -16810.264} C_VEL
LIN {X 0,Y 291.467,Z 162.178,A -85,B 0,C 180,E1 -16814.682,E2 -16814.682} C_VEL
LIN {X 0,Y 291.519,Z 162.17,A -85,B 0,C 180,E1 -16818.88,E2 -16818.88} C_VEL
LIN {X 0,Y 291.644,Z 162.155,A -85,B 0,C 180,E1 -16821.686,E2 -16821.686} C_VEL
LIN {X 0,Y 291.682,Z 162.209,A -85,B 0,C 180,E1 -16823.862,E2 -16823.862} C_VEL
LIN {X 0,Y 292.305,Z 165.732,A -85,B 0,C 180,E1 -16825.042,E2 -16825.042} C_VEL
LIN {X 0,Y 299.082,Z 182.363,A -85,B 0,C 180,E1 -16826.083,E2 -16826.083} C_VEL
LIN {X 0,Y 303.181,Z 194.228,A -85,B 0,C 180,E1 -16826.734,E2 -16826.734} C_VEL
LIN {X 0,Y 303.859,Z 198.192,A -85,B 0,C 180,E1 -16826.892,E2 -16826.892} C_VEL
LIN {X 0,Y 301.743,Z 272.982,A -85,B 0,C 180,E1 -16828.707,E2 -16828.707} C_VEL
LIN {X 0,Y 300.971,Z 286.205,A -85,B 0,C 180,E1 -16829.289,E2 -16829.289} C_VEL
LIN {X 0,Y 300.074,Z 298.323,A -85,B 0,C 180,E1 -16830.084,E2 -16830.084} C_VEL
LIN {X 0,Y 298.891,Z 310.598,A -85,B 0,C 180,E1 -16831.179,E2 -16831.179} C_VEL
LIN {X 0,Y 297.408,Z 322.323,A -85,B 0,C 180,E1 -16832.539,E2 -16832.539} C_VEL
LIN {X 0,Y 295.926,Z 332.945,A -85,B 0,C 180,E1 -16834.101,E2 -16834.101} C_VEL
LIN {X 0,Y 294.508,Z 342.264,A -85,B 0,C 180,E1 -16835.821,E2 -16835.821} C_VEL
LIN {X 0,Y 293.027,Z 351.42,A -85,B 0,C 180,E1 -16837.927,E2 -16837.927} C_VEL
LIN {X 0,Y 291.819,Z 358.744,A -85,B 0,C 180,E1 -16840.055,E2 -16840.055} C_VEL
LIN {X 0,Y 291.03,Z 363.697,A -85,B 0,C 180,E1 -16841.845,E2 -16841.845} C_VEL
LIN {X 0,Y 290.226,Z 369.145,A -85,B 0,C 180,E1 -16844.396,E2 -16844.396} C_VEL
LIN {X 0,Y 289.634,Z 372.995,A -85,B 0,C 180,E1 -16846.928,E2 -16846.928} C_VEL
LIN {X 0,Y 289.412,Z 374.832,A -85,B 0,C 180,E1 -16848.73,E2 -16848.73} C_VEL
LIN {X 0,Y 289.246,Z 376.32,A -85,B 0,C 180,E1 -16851.375,E2 -16851.375} C_VEL
LIN {X 0,Y 289.269,Z 376.521,A -85,B 0,C 180,E1 -16852.875,E2 -16852.875} C_VEL
LIN {X 0,Y 289.349,Z 376.242,A -85,B 0,C 180,E1 -16854.388,E2 -16854.388} C_VEL
LIN {X 0,Y 289.578,Z 375.394,A -85,B 0,C 180,E1 -16856.109,E2 -16856.109} C_VEL
LIN {X 0,Y 289.815,Z 374.287,A -85,B 0,C 180,E1 -16857.435,E2 -16857.435} C_VEL
LIN {X 0,Y 290.282,Z 372.052,A -85,B 0,C 180,E1 -16859.359,E2 -16859.359} C_VEL
LIN {X 0,Y 290.873,Z 368.922,A -85,B 0,C 180,E1 -16861.297,E2 -16861.297} C_VEL
LIN {X 0,Y 291.931,Z 363.932,A -85,B 0,C 180,E1 -16863.622,E2 -16863.622} C_VEL
LIN {X 0,Y 293.3,Z 357.288,A -85,B 0,C 180,E1 -16865.962,E2 -16865.962} C_VEL
LIN {X 0,Y 294.959,Z 349.301,A -85,B 0,C 180,E1 -16868.162,E2 -16868.162} C_VEL
LIN {X 0,Y 296.771,Z 340.129,A -85,B 0,C 180,E1 -16870.14,E2 -16870.14} C_VEL
LIN {X 0,Y 298.662,Z 329.94,A -85,B 0,C 180,E1 -16871.89,E2 -16871.89} C_VEL
LIN {X 0,Y 300.325,Z 319.571,A -85,B 0,C 180,E1 -16873.313,E2 -16873.313} C_VEL
LIN {X 0,Y 301.96,Z 308.317,A -85,B 0,C 180,E1 -16874.519,E2 -16874.519} C_VEL
LIN {X 0,Y 303.301,Z 295.785,A -85,B 0,C 180,E1 -16875.559,E2 -16875.559} C_VEL
LIN {X 0,Y 304.315,Z 282.872,A -85,B 0,C 180,E1 -16876.326,E2 -16876.326} C_VEL
LIN {X 0,Y 305.037,Z 269.81,A -85,B 0,C 180,E1 -16876.813,E2 -16876.813} C_VEL
LIN {X 0,Y 307.282,Z 199.514,A -85,B 0,C 180,E1 -16878.506,E2 -16878.506} C_VEL
LIN {X 0,Y 300.698,Z 183.378,A -85,B 0,C 180,E1 -16879.677,E2 -16879.677} C_VEL
LIN {X 0,Y 293.896,Z 169.479,A -85,B 0,C 180,E1 -16880.883,E2 -16880.883} C_VEL
LIN {X 0,Y 292.461,Z 166.397,A -85,B 0,C 180,E1 -16881.181,E2 -16881.181} C_VEL
LIN {X 0,Y 291.429,Z 162.19,A -85,B 0,C 180,E1 -16882.857,E2 -16882.857} C_VEL
LIN {X 0,Y 291.411,Z 162.19,A -85,B 0,C 180,E1 -16883.134,E2 -16883.134} C_VEL
LIN {X 0,Y 290.676,Z 162.282,A -85,B 0,C 180,E1 -16884.288,E2 -16884.288} C_VEL
LIN {X 0,Y 287.783,Z 162.638,A -85,B 0,C 180,E1 -16886.167,E2 -16886.167} C_VEL
LIN {X 0,Y 285.377,Z 162.937,A -85,B 0,C 180,E1 -16887.692,E2 -16887.692} C_VEL
LIN {X 0,Y 284.363,Z 163.063,A -85,B 0,C 180,E1 -16888.874,E2 -16888.874} C_VEL
LIN {X 0,Y 284.287,Z 163.069,A -85,B 0,C 180,E1 -16889.275,E2 -16889.275} C_VEL
LIN {X 0,Y 284.376,Z 163.063,A -85,B 0,C 180,E1 -16893.588,E2 -16893.588} C_VEL
LIN {X 0,Y 284.365,Z 163.064,A -85,B 0,C 180,E1 -16896.708,E2 -16896.708} C_VEL
LIN {X 0,Y 284.385,Z 163.062,A -85,B 0,C 180,E1 -16901.262,E2 -16901.262} C_VEL
LIN {X 0,Y 284.463,Z 163.047,A -85,B 0,C 180,E1 -16905.698,E2 -16905.698} C_VEL
LIN {X 0,Y 284.514,Z 163.04,A -85,B 0,C 180,E1 -16910.044,E2 -16910.044} C_VEL
LIN {X 0,Y 284.646,Z 163.027,A -85,B 0,C 180,E1 -16912.91,E2 -16912.91} C_VEL
LIN {X 0,Y 284.852,Z 162.999,A -85,B 0,C 180,E1 -16918.587,E2 -16918.587} C_VEL
LIN {X 0,Y 284.847,Z 162.988,A -85,B 0,C 180,E1 -16921.415,E2 -16921.415} C_VEL
LIN {X 0,Y 284.645,Z 163.02,A -85,B 0,C 180,E1 -16927.093,E2 -16927.093} C_VEL
LIN {X 0,Y 284.516,Z 163.033,A -85,B 0,C 180,E1 -16929.958,E2 -16929.958} C_VEL
LIN {X 0,Y 284.451,Z 163.051,A -85,B 0,C 180,E1 -16934.305,E2 -16934.305} C_VEL
LIN {X 0,Y 284.328,Z 163.067,A -85,B 0,C 180,E1 -16938.745,E2 -16938.745} C_VEL
LIN {X 0,Y 284.3,Z 163.06,A -85,B 0,C 180,E1 -16941.766,E2 -16941.766} C_VEL
LIN {X 0,Y 284.285,Z 163.072,A -85,B 0,C 180,E1 -16944.853,E2 -16944.853} C_VEL
LIN {X 0,Y 284.283,Z 163.074,A -85,B 0,C 180,E1 -16948.017,E2 -16948.017} C_VEL
LIN {X 0,Y 284.287,Z 163.065,A -85,B 0,C 180,E1 -16951.277,E2 -16951.277} C_VEL
LIN {X 0,Y 284.339,Z 163.062,A -85,B 0,C 180,E1 -16955.347,E2 -16955.347} C_VEL
LIN {X 0,Y 284.267,Z 163.069,A -85,B 0,C 180,E1 -16958.177,E2 -16958.177} C_VEL
LIN {X 0,Y 284.239,Z 163.082,A -85,B 0,C 180,E1 -16962.118,E2 -16962.118} C_VEL
LIN {X 0,Y 284.24,Z 163.083,A -85,B 0,C 180,E1 -16966.186,E2 -16966.186} C_VEL
LIN {X 0,Y 284.258,Z 163.081,A -85,B 0,C 180,E1 -16970.037,E2 -16970.037} C_VEL
LIN {X 0,Y 284.362,Z 163.242,A -85,B 0,C 180,E1 -16973.178,E2 -16973.178} C_VEL
LIN {X 0,Y 286.602,Z 172.066,A -85,B 0,C 180,E1 -16976.487,E2 -16976.487} C_VEL
LIN {X 0,Y 288.674,Z 181.113,A -85,B 0,C 180,E1 -16979.657,E2 -16979.657} C_VEL
LIN {X 0,Y 289.258,Z 183.807,A -85,B 0,C 180,E1 -16980.491,E2 -16980.491} C_VEL
LIN {X 0,Y 294.402,Z 196.05,A -85,B 0,C 180,E1 -16981.482,E2 -16981.482} C_VEL
LIN {X 0,Y 298.183,Z 217.157,A -85,B 0,C 180,E1 -16982.522,E2 -16982.522} C_VEL
LIN {X 0,Y 300.11,Z 232.094,A -85,B 0,C 180,E1 -16983.154,E2 -16983.154} C_VEL
LIN {X 0,Y 298.186,Z 293.332,A -85,B 0,C 180,E1 -16984.704,E2 -16984.704} C_VEL
LIN {X 0,Y 297.047,Z 307.002,A -85,B 0,C 180,E1 -16985.308,E2 -16985.308} C_VEL
LIN {X 0,Y 295.538,Z 319.783,A -85,B 0,C 180,E1 -16986.155,E2 -16986.155} C_VEL
LIN {X 0,Y 293.742,Z 332.279,A -85,B 0,C 180,E1 -16987.307,E2 -16987.307} C_VEL
LIN {X 0,Y 291.884,Z 343.47,A -85,B 0,C 180,E1 -16988.643,E2 -16988.643} C_VEL
LIN {X 0,Y 289.922,Z 353.574,A -85,B 0,C 180,E1 -16990.161,E2 -16990.161} C_VEL
LIN {X 0,Y 288.225,Z 362.567,A -85,B 0,C 180,E1 -16991.854,E2 -16991.854} C_VEL
LIN {X 0,Y 286.417,Z 371.65,A -85,B 0,C 180,E1 -16993.976,E2 -16993.976} C_VEL
LIN {X 0,Y 284.916,Z 378.854,A -85,B 0,C 180,E1 -16996.084,E2 -16996.084} C_VEL
LIN {X 0,Y 283.89,Z 383.731,A -85,B 0,C 180,E1 -16997.853,E2 -16997.853} C_VEL
LIN {X 0,Y 283.138,Z 388.487,A -85,B 0,C 180,E1 -16999.994,E2 -16999.994} C_VEL
LIN {X 0,Y 282.645,Z 392.135,A -85,B 0,C 180,E1 -17002.14,E2 -17002.14} C_VEL
LIN {X 0,Y 282.348,Z 395.165,A -85,B 0,C 180,E1 -17004.663,E2 -17004.663} C_VEL
LIN {X 0,Y 282.378,Z 396.859,A -85,B 0,C 180,E1 -17007.147,E2 -17007.147} C_VEL
LIN {X 0,Y 282.373,Z 397.269,A -85,B 0,C 180,E1 -17008.574,E2 -17008.574} C_VEL
LIN {X 0,Y 282.414,Z 397.291,A -85,B 0,C 180,E1 -17010,E2 -17010} C_VEL
LIN {X 0,Y 282.382,Z 396.919,A -85,B 0,C 180,E1 -17011.426,E2 -17011.426} C_VEL
LIN {X 0,Y 282.379,Z 396.121,A -85,B 0,C 180,E1 -17012.854,E2 -17012.854} C_VEL
LIN {X 0,Y 282.348,Z 393.724,A -85,B 0,C 180,E1 -17015.336,E2 -17015.336} C_VEL
LIN {X 0,Y 282.643,Z 389.938,A -85,B 0,C 180,E1 -17017.861,E2 -17017.861} C_VEL
LIN {X 0,Y 283.091,Z 385.536,A -85,B 0,C 180,E1 -17020.008,E2 -17020.008} C_VEL
LIN {X 0,Y 283.784,Z 379.92,A -85,B 0,C 180,E1 -17022.152,E2 -17022.152} C_VEL
LIN {X 0,Y 284.976,Z 372.906,A -85,B 0,C 180,E1 -17024.278,E2 -17024.278} C_VEL
LIN {X 0,Y 286.385,Z 364.216,A -85,B 0,C 180,E1 -17026.365,E2 -17026.365} C_VEL
LIN {X 0,Y 287.806,Z 354.058,A -85,B 0,C 180,E1 -17028.325,E2 -17028.325} C_VEL
LIN {X 0,Y 289.485,Z 343.862,A -85,B 0,C 180,E1 -17029.87,E2 -17029.87} C_VEL
LIN {X 0,Y 291.099,Z 332.536,A -85,B 0,C 180,E1 -17031.232,E2 -17031.232} C_VEL
LIN {X 0,Y 292.516,Z 320.806,A -85,B 0,C 180,E1 -17032.329,E2 -17032.329} C_VEL
LIN {X 0,Y 293.848,Z 308.076,A -85,B 0,C 180,E1 -17033.197,E2 -17033.197} C_VEL
LIN {X 0,Y 294.744,Z 294.572,A -85,B 0,C 180,E1 -17033.82,E2 -17033.82} C_VEL
LIN {X 0,Y 295.907,Z 255.625,A -85,B 0,C 180,E1 -17034.817,E2 -17034.817} C_VEL
LIN {X 0,Y 296.447,Z 229.32,A -85,B 0,C 180,E1 -17035.474,E2 -17035.474} C_VEL
LIN {X 0,Y 290.808,Z 191.676,A -85,B 0,C 180,E1 -17036.973,E2 -17036.973} C_VEL
LIN {X 0,Y 289.396,Z 186.5,A -85,B 0,C 180,E1 -17037.243,E2 -17037.243} C_VEL
LIN {X 0,Y 288.892,Z 184.708,A -85,B 0,C 180,E1 -17037.361,E2 -17037.361} C_VEL
LIN {X 0,Y 286.634,Z 173.335,A -85,B 0,C 180,E1 -17040.991,E2 -17040.991} C_VEL
LIN {X 0,Y 284.353,Z 163.066,A -85,B 0,C 180,E1 -17044.486,E2 -17044.486} C_VEL
LIN {X 0,Y 284.271,Z 163.072,A -85,B 0,C 180,E1 -17048.176,E2 -17048.176} C_VEL
LIN {X 0,Y 284.241,Z 163.072,A -85,B 0,C 180,E1 -17052.117,E2 -17052.117} C_VEL
LIN {X 0,Y 284.242,Z 163.077,A -85,B 0,C 180,E1 -17056.185,E2 -17056.185} C_VEL
LIN {X 0,Y 284.288,Z 163.072,A -85,B 0,C 180,E1 -17060.029,E2 -17060.029} C_VEL
LIN {X 0,Y 284.331,Z 163.068,A -85,B 0,C 180,E1 -17063.613,E2 -17063.613} C_VEL
LIN {X 0,Y 284.311,Z 163.072,A -85,B 0,C 180,E1 -17067.19,E2 -17067.19} C_VEL
LIN {X 0,Y 284.342,Z 163.065,A -85,B 0,C 180,E1 -17070.373,E2 -17070.373} C_VEL
LIN {X 0,Y 284.31,Z 163.069,A -85,B 0,C 180,E1 -17073.579,E2 -17073.579} C_VEL
LIN {X 0,Y 284.332,Z 163.07,A -85,B 0,C 180,E1 -17076.703,E2 -17076.703} C_VEL
LIN {X 0,Y 284.327,Z 163.066,A -85,B 0,C 180,E1 -17081.255,E2 -17081.255} C_VEL
LIN {X 0,Y 284.423,Z 163.053,A -85,B 0,C 180,E1 -17085.693,E2 -17085.693} C_VEL
LIN {X 0,Y 284.518,Z 163.04,A -85,B 0,C 180,E1 -17090.042,E2 -17090.042} C_VEL
LIN {X 0,Y 284.646,Z 163.02,A -85,B 0,C 180,E1 -17092.908,E2 -17092.908} C_VEL
LIN {X 0,Y 284.841,Z 163.003,A -85,B 0,C 180,E1 -17098.585,E2 -17098.585} C_VEL
LIN {X 0,Y 284.841,Z 162.997,A -85,B 0,C 180,E1 -17101.413,E2 -17101.413} C_VEL
LIN {X 0,Y 284.644,Z 163.024,A -85,B 0,C 180,E1 -17107.09,E2 -17107.09} C_VEL
LIN {X 0,Y 284.516,Z 163.047,A -85,B 0,C 180,E1 -17109.956,E2 -17109.956} C_VEL
LIN {X 0,Y 284.419,Z 163.046,A -85,B 0,C 180,E1 -17114.305,E2 -17114.305} C_VEL
LIN {X 0,Y 284.318,Z 163.064,A -85,B 0,C 180,E1 -17118.743,E2 -17118.743} C_VEL
LIN {X 0,Y 284.297,Z 163.073,A -85,B 0,C 180,E1 -17121.764,E2 -17121.764} C_VEL
LIN {X 0,Y 284.282,Z 163.068,A -85,B 0,C 180,E1 -17124.85,E2 -17124.85} C_VEL
LIN {X 0,Y 284.259,Z 163.068,A -85,B 0,C 180,E1 -17128.017,E2 -17128.017} C_VEL
LIN {X 0,Y 284.277,Z 163.073,A -85,B 0,C 180,E1 -17131.275,E2 -17131.275} C_VEL
LIN {X 0,Y 284.335,Z 163.066,A -85,B 0,C 180,E1 -17135.345,E2 -17135.345} C_VEL
LIN {X 0,Y 284.264,Z 163.065,A -85,B 0,C 180,E1 -17138.175,E2 -17138.175} C_VEL
LIN {X 0,Y 284.234,Z 163.078,A -85,B 0,C 180,E1 -17142.116,E2 -17142.116} C_VEL
LIN {X 0,Y 284.234,Z 163.074,A -85,B 0,C 180,E1 -17146.184,E2 -17146.184} C_VEL
LIN {X 0,Y 284.279,Z 163.072,A -85,B 0,C 180,E1 -17150.028,E2 -17150.028} C_VEL
LIN {X 0,Y 284.316,Z 163.066,A -85,B 0,C 180,E1 -17153.611,E2 -17153.611} C_VEL
LIN {X 0,Y 284.301,Z 163.072,A -85,B 0,C 180,E1 -17157.189,E2 -17157.189} C_VEL
LIN {X 0,Y 284.331,Z 163.067,A -85,B 0,C 180,E1 -17160.372,E2 -17160.372} C_VEL
LIN {X 0,Y 284.291,Z 163.071,A -85,B 0,C 180,E1 -17163.577,E2 -17163.577} C_VEL
LIN {X 0,Y 284.301,Z 163.067,A -85,B 0,C 180,E1 -17166.701,E2 -17166.701} C_VEL
LIN {X 0,Y 284.327,Z 163.068,A -85,B 0,C 180,E1 -17169.927,E2 -17169.927} C_VEL
LIN {X 0,Y 284.408,Z 163.058,A -85,B 0,C 180,E1 -17174.516,E2 -17174.516} C_VEL
LIN {X 0,Y 284.456,Z 163.05,A -85,B 0,C 180,E1 -17178.6,E2 -17178.6} C_VEL
LIN {X 0,Y 284.601,Z 163.031,A -85,B 0,C 180,E1 -17181.479,E2 -17181.479} C_VEL
LIN {X 0,Y 284.663,Z 163.216,A -85,B 0,C 180,E1 -17183.443,E2 -17183.443} C_VEL
LIN {X 0,Y 285.158,Z 165.94,A -85,B 0,C 180,E1 -17184.388,E2 -17184.388} C_VEL
LIN {X 0,Y 292.966,Z 185.117,A -85,B 0,C 180,E1 -17185.633,E2 -17185.633} C_VEL
LIN {X 0,Y 296.919,Z 196.854,A -85,B 0,C 180,E1 -17186.289,E2 -17186.289} C_VEL
LIN {X 0,Y 297.286,Z 200.383,A -85,B 0,C 180,E1 -17186.414,E2 -17186.414} C_VEL
LIN {X 0,Y 295.13,Z 273.113,A -85,B 0,C 180,E1 -17188.214,E2 -17188.214} C_VEL
LIN {X 0,Y 294.34,Z 286.268,A -85,B 0,C 180,E1 -17188.803,E2 -17188.803} C_VEL
LIN {X 0,Y 293.381,Z 298.989,A -85,B 0,C 180,E1 -17189.657,E2 -17189.657} C_VEL
LIN {X 0,Y 292.253,Z 310.34,A -85,B 0,C 180,E1 -17190.689,E2 -17190.689} C_VEL
LIN {X 0,Y 290.697,Z 322.171,A -85,B 0,C 180,E1 -17192.078,E2 -17192.078} C_VEL
LIN {X 0,Y 289.226,Z 332.276,A -85,B 0,C 180,E1 -17193.576,E2 -17193.576} C_VEL
LIN {X 0,Y 287.823,Z 341.423,A -85,B 0,C 180,E1 -17195.253,E2 -17195.253} C_VEL
LIN {X 0,Y 286.242,Z 350.771,A -85,B 0,C 180,E1 -17197.406,E2 -17197.406} C_VEL
LIN {X 0,Y 284.986,Z 357.897,A -85,B 0,C 180,E1 -17199.457,E2 -17199.457} C_VEL
LIN {X 0,Y 284.112,Z 363.349,A -85,B 0,C 180,E1 -17201.414,E2 -17201.414} C_VEL
LIN {X 0,Y 283.33,Z 368.249,A -85,B 0,C 180,E1 -17203.63,E2 -17203.63} C_VEL
LIN {X 0,Y 282.778,Z 371.971,A -85,B 0,C 180,E1 -17205.866,E2 -17205.866} C_VEL
LIN {X 0,Y 282.489,Z 373.832,A -85,B 0,C 180,E1 -17207.37,E2 -17207.37} C_VEL
LIN {X 0,Y 282.31,Z 375.263,A -85,B 0,C 180,E1 -17208.92,E2 -17208.92} C_VEL
LIN {X 0,Y 282.181,Z 376.21,A -85,B 0,C 180,E1 -17210.407,E2 -17210.407} C_VEL
LIN {X 0,Y 282.174,Z 376.792,A -85,B 0,C 180,E1 -17212.851,E2 -17212.851} C_VEL
LIN {X 0,Y 282.328,Z 376.333,A -85,B 0,C 180,E1 -17215.035,E2 -17215.035} C_VEL
LIN {X 0,Y 282.563,Z 375.41,A -85,B 0,C 180,E1 -17216.596,E2 -17216.596} C_VEL
LIN {X 0,Y 282.867,Z 374.018,A -85,B 0,C 180,E1 -17218.168,E2 -17218.168} C_VEL
LIN {X 0,Y 283.529,Z 370.949,A -85,B 0,C 180,E1 -17220.54,E2 -17220.54} C_VEL
LIN {X 0,Y 284.489,Z 366.577,A -85,B 0,C 180,E1 -17222.921,E2 -17222.921} C_VEL
LIN {X 0,Y 285.687,Z 361.039,A -85,B 0,C 180,E1 -17225.185,E2 -17225.185} C_VEL
LIN {X 0,Y 287.144,Z 354.504,A -85,B 0,C 180,E1 -17227.284,E2 -17227.284} C_VEL
LIN {X 0,Y 288.788,Z 346.867,A -85,B 0,C 180,E1 -17229.252,E2 -17229.252} C_VEL
LIN {X 0,Y 290.577,Z 338.193,A -85,B 0,C 180,E1 -17231.059,E2 -17231.059} C_VEL
LIN {X 0,Y 292.483,Z 328.008,A -85,B 0,C 180,E1 -17232.751,E2 -17232.751} C_VEL
LIN {X 0,Y 294.366,Z 316.577,A -85,B 0,C 180,E1 -17234.256,E2 -17234.256} C_VEL
LIN {X 0,Y 295.981,Z 305.158,A -85,B 0,C 180,E1 -17235.426,E2 -17235.426} C_VEL
LIN {X 0,Y 297.263,Z 292.715,A -85,B 0,C 180,E1 -17236.39,E2 -17236.39} C_VEL
LIN {X 0,Y 298.23,Z 279.54,A -85,B 0,C 180,E1 -17237.112,E2 -17237.112} C_VEL
LIN {X 0,Y 298.922,Z 266.179,A -85,B 0,C 180,E1 -17237.544,E2 -17237.544} C_VEL
LIN {X 0,Y 301.055,Z 201.312,A -85,B 0,C 180,E1 -17239.131,E2 -17239.131} C_VEL
LIN {X 0,Y 295.108,Z 186.688,A -85,B 0,C 180,E1 -17240.231,E2 -17240.231} C_VEL
LIN {X 0,Y 288.557,Z 173.3,A -85,B 0,C 180,E1 -17241.44,E2 -17241.44} C_VEL
LIN {X 0,Y 285.303,Z 166.719,A -85,B 0,C 180,E1 -17242.096,E2 -17242.096} C_VEL
LIN {X 0,Y 284.352,Z 163.073,A -85,B 0,C 180,E1 -17243.619,E2 -17243.619} C_VEL
LIN {X 0,Y 284.305,Z 163.073,A -85,B 0,C 180,E1 -17247.191,E2 -17247.191} C_VEL
LIN {X 0,Y 284.287,Z 163.069,A -85,B 0,C 180,E1 -17249.275,E2 -17249.275} C_VEL
LIN {X 0,Y 283.634,Z 163.152,A -85,B 0,C 180,E1 -17250.458,E2 -17250.458} C_VEL
LIN {X 0,Y 280.785,Z 163.509,A -85,B 0,C 180,E1 -17252.385,E2 -17252.385} C_VEL
LIN {X 0,Y 278.377,Z 163.813,A -85,B 0,C 180,E1 -17253.95,E2 -17253.95} C_VEL
LIN {X 0,Y 277.372,Z 163.934,A -85,B 0,C 180,E1 -17255.164,E2 -17255.164} C_VEL
LIN {X 0,Y 277.305,Z 163.94,A -85,B 0,C 180,E1 -17255.574,E2 -17255.574} C_VEL
LIN {X 0,Y 277.343,Z 163.935,A -85,B 0,C 180,E1 -17259.652,E2 -17259.652} C_VEL
LIN {X 0,Y 277.411,Z 163.929,A -85,B 0,C 180,E1 -17264.302,E2 -17264.302} C_VEL
LIN {X 0,Y 277.43,Z 163.925,A -85,B 0,C 180,E1 -17268.309,E2 -17268.309} C_VEL
LIN {X 0,Y 277.57,Z 163.898,A -85,B 0,C 180,E1 -17271.263,E2 -17271.263} C_VEL
LIN {X 0,Y 277.547,Z 163.909,A -85,B 0,C 180,E1 -17274.188,E2 -17274.188} C_VEL
LIN {X 0,Y 277.818,Z 163.875,A -85,B 0,C 180,E1 -17278.552,E2 -17278.552} C_VEL
LIN {X 0,Y 277.813,Z 163.864,A -85,B 0,C 180,E1 -17281.451,E2 -17281.451} C_VEL
LIN {X 0,Y 277.603,Z 163.898,A -85,B 0,C 180,E1 -17287.273,E2 -17287.273} C_VEL
LIN {X 0,Y 277.457,Z 163.909,A -85,B 0,C 180,E1 -17290.214,E2 -17290.214} C_VEL
LIN {X 0,Y 277.399,Z 163.927,A -85,B 0,C 180,E1 -17294.677,E2 -17294.677} C_VEL
LIN {X 0,Y 277.283,Z 163.946,A -85,B 0,C 180,E1 -17299.239,E2 -17299.239} C_VEL
LIN {X 0,Y 277.258,Z 163.949,A -85,B 0,C 180,E1 -17303.928,E2 -17303.928} C_VEL
LIN {X 0,Y 277.269,Z 163.942,A -85,B 0,C 180,E1 -17307.482,E2 -17307.482} C_VEL
LIN {X 0,Y 277.25,Z 163.939,A -85,B 0,C 180,E1 -17310.474,E2 -17310.474} C_VEL
LIN {X 0,Y 277.248,Z 163.943,A -85,B 0,C 180,E1 -17313.897,E2 -17313.897} C_VEL
LIN {X 0,Y 277.235,Z 163.946,A -85,B 0,C 180,E1 -17317.476,E2 -17317.476} C_VEL
LIN {X 0,Y 277.179,Z 163.957,A -85,B 0,C 180,E1 -17321.243,E2 -17321.243} C_VEL
LIN {X 0,Y 277.176,Z 163.966,A -85,B 0,C 180,E1 -17325.233,E2 -17325.233} C_VEL
LIN {X 0,Y 277.179,Z 163.961,A -85,B 0,C 180,E1 -17328.758,E2 -17328.758} C_VEL
LIN {X 0,Y 277.267,Z 164.032,A -85,B 0,C 180,E1 -17332.307,E2 -17332.307} C_VEL
LIN {X 0,Y 279.731,Z 173.493,A -85,B 0,C 180,E1 -17336.008,E2 -17336.008} C_VEL
LIN {X 0,Y 281.974,Z 183.321,A -85,B 0,C 180,E1 -17339.523,E2 -17339.523} C_VEL
LIN {X 0,Y 288.592,Z 198.627,A -85,B 0,C 180,E1 -17340.853,E2 -17340.853} C_VEL
LIN {X 0,Y 292.02,Z 217.973,A -85,B 0,C 180,E1 -17341.842,E2 -17341.842} C_VEL
LIN {X 0,Y 293.937,Z 232.358,A -85,B 0,C 180,E1 -17342.479,E2 -17342.479} C_VEL
LIN {X 0,Y 291.939,Z 293.125,A -85,B 0,C 180,E1 -17344.049,E2 -17344.049} C_VEL
LIN {X 0,Y 290.715,Z 307.186,A -85,B 0,C 180,E1 -17344.685,E2 -17344.685} C_VEL
LIN {X 0,Y 289.262,Z 319.312,A -85,B 0,C 180,E1 -17345.509,E2 -17345.509} C_VEL
LIN {X 0,Y 287.463,Z 331.061,A -85,B 0,C 180,E1 -17346.592,E2 -17346.592} C_VEL
LIN {X 0,Y 285.536,Z 342.407,A -85,B 0,C 180,E1 -17347.954,E2 -17347.954} C_VEL
LIN {X 0,Y 283.462,Z 352.678,A -85,B 0,C 180,E1 -17349.5,E2 -17349.5} C_VEL
LIN {X 0,Y 281.797,Z 361.096,A -85,B 0,C 180,E1 -17351.082,E2 -17351.082} C_VEL
LIN {X 0,Y 279.849,Z 370.254,A -85,B 0,C 180,E1 -17353.214,E2 -17353.214} C_VEL
LIN {X 0,Y 278.249,Z 377.663,A -85,B 0,C 180,E1 -17355.37,E2 -17355.37} C_VEL
LIN {X 0,Y 276.918,Z 383.625,A -85,B 0,C 180,E1 -17357.542,E2 -17357.542} C_VEL
LIN {X 0,Y 276.13,Z 388.348,A -85,B 0,C 180,E1 -17359.738,E2 -17359.738} C_VEL
LIN {X 0,Y 275.575,Z 391.966,A -85,B 0,C 180,E1 -17361.937,E2 -17361.937} C_VEL
LIN {X 0,Y 275.252,Z 395.138,A -85,B 0,C 180,E1 -17364.747,E2 -17364.747} C_VEL
LIN {X 0,Y 275.284,Z 396.619,A -85,B 0,C 180,E1 -17367.073,E2 -17367.073} C_VEL
LIN {X 0,Y 275.296,Z 397.016,A -85,B 0,C 180,E1 -17368.537,E2 -17368.537} C_VEL
LIN {X 0,Y 275.333,Z 397.024,A -85,B 0,C 180,E1 -17370,E2 -17370} C_VEL
LIN {X 0,Y 275.304,Z 396.638,A -85,B 0,C 180,E1 -17371.463,E2 -17371.463} C_VEL
LIN {X 0,Y 275.285,Z 395.812,A -85,B 0,C 180,E1 -17372.927,E2 -17372.927} C_VEL
LIN {X 0,Y 275.252,Z 393.655,A -85,B 0,C 180,E1 -17375.253,E2 -17375.253} C_VEL
LIN {X 0,Y 275.571,Z 389.566,A -85,B 0,C 180,E1 -17378.064,E2 -17378.064} C_VEL
LIN {X 0,Y 276.062,Z 385.129,A -85,B 0,C 180,E1 -17380.266,E2 -17380.266} C_VEL
LIN {X 0,Y 276.81,Z 379.474,A -85,B 0,C 180,E1 -17382.463,E2 -17382.463} C_VEL
LIN {X 0,Y 278.047,Z 372.4,A -85,B 0,C 180,E1 -17384.641,E2 -17384.641} C_VEL
LIN {X 0,Y 279.463,Z 364.07,A -85,B 0,C 180,E1 -17386.687,E2 -17386.687} C_VEL
LIN {X 0,Y 280.859,Z 354.417,A -85,B 0,C 180,E1 -17388.606,E2 -17388.606} C_VEL
LIN {X 0,Y 282.588,Z 344.409,A -85,B 0,C 180,E1 -17390.187,E2 -17390.187} C_VEL
LIN {X 0,Y 284.218,Z 333.271,A -85,B 0,C 180,E1 -17391.582,E2 -17391.582} C_VEL
LIN {X 0,Y 285.814,Z 320.8,A -85,B 0,C 180,E1 -17392.786,E2 -17392.786} C_VEL
LIN {X 0,Y 287.191,Z 308.202,A -85,B 0,C 180,E1 -17393.672,E2 -17393.672} C_VEL
LIN {X 0,Y 288.108,Z 294.883,A -85,B 0,C 180,E1 -17394.308,E2 -17394.308} C_VEL
LIN {X 0,Y 288.992,Z 268.955,A -85,B 0,C 180,E1 -17395.006,E2 -17395.006} C_VEL
LIN {X 0,Y 289.934,Z 230.233,A -85,B 0,C 180,E1 -17395.986,E2 -17395.986} C_VEL
LIN {X 0,Y 284.295,Z 192.592,A -85,B 0,C 180,E1 -17397.535,E2 -17397.535} C_VEL
LIN {X 0,Y 281.672,Z 184.4,A -85,B 0,C 180,E1 -17398.046,E2 -17398.046} C_VEL
LIN {X 0,Y 279.276,Z 172.736,A -85,B 0,C 180,E1 -17401.902,E2 -17401.902} C_VEL
LIN {X 0,Y 277.291,Z 163.944,A -85,B 0,C 180,E1 -17404.991,E2 -17404.991} C_VEL
LIN {X 0,Y 277.196,Z 163.955,A -85,B 0,C 180,E1 -17409.335,E2 -17409.335} C_VEL
LIN {X 0,Y 277.196,Z 163.952,A -85,B 0,C 180,E1 -17413.201,E2 -17413.201} C_VEL
LIN {X 0,Y 277.197,Z 163.959,A -85,B 0,C 180,E1 -17417.33,E2 -17417.33} C_VEL
LIN {X 0,Y 277.26,Z 163.948,A -85,B 0,C 180,E1 -17421.795,E2 -17421.795} C_VEL
LIN {X 0,Y 277.284,Z 163.945,A -85,B 0,C 180,E1 -17424.34,E2 -17424.34} C_VEL
LIN {X 0,Y 277.245,Z 163.949,A -85,B 0,C 180,E1 -17427.835,E2 -17427.835} C_VEL
LIN {X 0,Y 277.244,Z 163.951,A -85,B 0,C 180,E1 -17431.206,E2 -17431.206} C_VEL
LIN {X 0,Y 277.251,Z 163.95,A -85,B 0,C 180,E1 -17434.472,E2 -17434.472} C_VEL
LIN {X 0,Y 277.263,Z 163.946,A -85,B 0,C 180,E1 -17437.652,E2 -17437.652} C_VEL
LIN {X 0,Y 277.284,Z 163.947,A -85,B 0,C 180,E1 -17440.761,E2 -17440.761} C_VEL
LIN {X 0,Y 277.376,Z 163.932,A -85,B 0,C 180,E1 -17445.322,E2 -17445.322} C_VEL
LIN {X 0,Y 277.461,Z 163.918,A -85,B 0,C 180,E1 -17449.786,E2 -17449.786} C_VEL
LIN {X 0,Y 277.605,Z 163.897,A -85,B 0,C 180,E1 -17452.727,E2 -17452.727} C_VEL
LIN {X 0,Y 277.808,Z 163.879,A -85,B 0,C 180,E1 -17458.549,E2 -17458.549} C_VEL
LIN {X 0,Y 277.808,Z 163.873,A -85,B 0,C 180,E1 -17461.448,E2 -17461.448} C_VEL
LIN {X 0,Y 277.603,Z 163.901,A -85,B 0,C 180,E1 -17467.271,E2 -17467.271} C_VEL
LIN {X 0,Y 277.456,Z 163.924,A -85,B 0,C 180,E1 -17470.212,E2 -17470.212} C_VEL
LIN {X 0,Y 277.372,Z 163.921,A -85,B 0,C 180,E1 -17474.676,E2 -17474.676} C_VEL
LIN {X 0,Y 277.277,Z 163.941,A -85,B 0,C 180,E1 -17479.237,E2 -17479.237} C_VEL
LIN {X 0,Y 277.255,Z 163.946,A -85,B 0,C 180,E1 -17483.926,E2 -17483.926} C_VEL
LIN {X 0,Y 277.235,Z 163.94,A -85,B 0,C 180,E1 -17487.467,E2 -17487.467} C_VEL
LIN {X 0,Y 277.227,Z 163.947,A -85,B 0,C 180,E1 -17490.464,E2 -17490.464} C_VEL
LIN {X 0,Y 277.244,Z 163.949,A -85,B 0,C 180,E1 -17493.894,E2 -17493.894} C_VEL
LIN {X 0,Y 277.232,Z 163.942,A -85,B 0,C 180,E1 -17497.473,E2 -17497.473} C_VEL
LIN {X 0,Y 277.181,Z 163.958,A -85,B 0,C 180,E1 -17501.24,E2 -17501.24} C_VEL
LIN {X 0,Y 277.17,Z 163.957,A -85,B 0,C 180,E1 -17505.231,E2 -17505.231} C_VEL
LIN {X 0,Y 277.18,Z 163.954,A -85,B 0,C 180,E1 -17508.757,E2 -17508.757} C_VEL
LIN {X 0,Y 277.25,Z 163.95,A -85,B 0,C 180,E1 -17512.527,E2 -17512.527} C_VEL
LIN {X 0,Y 277.241,Z 163.946,A -85,B 0,C 180,E1 -17516.103,E2 -17516.103} C_VEL
LIN {X 0,Y 277.257,Z 163.946,A -85,B 0,C 180,E1 -17519.537,E2 -17519.537} C_VEL
LIN {X 0,Y 277.283,Z 163.947,A -85,B 0,C 180,E1 -17522.856,E2 -17522.856} C_VEL
LIN {X 0,Y 277.249,Z 163.946,A -85,B 0,C 180,E1 -17526.072,E2 -17526.072} C_VEL
LIN {X 0,Y 277.272,Z 163.948,A -85,B 0,C 180,E1 -17530.76,E2 -17530.76} C_VEL
LIN {X 0,Y 277.364,Z 163.932,A -85,B 0,C 180,E1 -17535.322,E2 -17535.322} C_VEL
LIN {X 0,Y 277.447,Z 163.924,A -85,B 0,C 180,E1 -17539.786,E2 -17539.786} C_VEL
LIN {X 0,Y 277.601,Z 163.976,A -85,B 0,C 180,E1 -17542.91,E2 -17542.91} C_VEL
LIN {X 0,Y 278.05,Z 166.085,A -85,B 0,C 180,E1 -17543.696,E2 -17543.696} C_VEL
LIN {X 0,Y 286.775,Z 187.531,A -85,B 0,C 180,E1 -17545.145,E2 -17545.145} C_VEL
LIN {X 0,Y 290.543,Z 198.711,A -85,B 0,C 180,E1 -17545.793,E2 -17545.793} C_VEL
LIN {X 0,Y 290.679,Z 203.512,A -85,B 0,C 180,E1 -17545.936,E2 -17545.936} C_VEL
LIN {X 0,Y 288.512,Z 273.775,A -85,B 0,C 180,E1 -17547.72,E2 -17547.72} C_VEL
LIN {X 0,Y 287.655,Z 287.313,A -85,B 0,C 180,E1 -17548.35,E2 -17548.35} C_VEL
LIN {X 0,Y 286.697,Z 299.642,A -85,B 0,C 180,E1 -17549.21,E2 -17549.21} C_VEL
LIN {X 0,Y 285.398,Z 311.704,A -85,B 0,C 180,E1 -17550.352,E2 -17550.352} C_VEL
LIN {X 0,Y 283.821,Z 323.323,A -85,B 0,C 180,E1 -17551.773,E2 -17551.773} C_VEL
LIN {X 0,Y 282.248,Z 333.605,A -85,B 0,C 180,E1 -17553.363,E2 -17553.363} C_VEL
LIN {X 0,Y 280.86,Z 342.257,A -85,B 0,C 180,E1 -17555.024,E2 -17555.024} C_VEL
LIN {X 0,Y 279.217,Z 351.511,A -85,B 0,C 180,E1 -17557.23,E2 -17557.23} C_VEL
LIN {X 0,Y 277.878,Z 358.99,A -85,B 0,C 180,E1 -17559.478,E2 -17559.478} C_VEL
LIN {X 0,Y 276.886,Z 364.818,A -85,B 0,C 180,E1 -17561.716,E2 -17561.716} C_VEL
LIN {X 0,Y 276.154,Z 369.304,A -85,B 0,C 180,E1 -17563.92,E2 -17563.92} C_VEL
LIN {X 0,Y 275.599,Z 372.894,A -85,B 0,C 180,E1 -17566.29,E2 -17566.29} C_VEL
LIN {X 0,Y 275.187,Z 375.68,A -85,B 0,C 180,E1 -17569.106,E2 -17569.106} C_VEL
LIN {X 0,Y 275.087,Z 376.667,A -85,B 0,C 180,E1 -17570.957,E2 -17570.957} C_VEL
LIN {X 0,Y 275.085,Z 377.037,A -85,B 0,C 180,E1 -17573.115,E2 -17573.115} C_VEL
LIN {X 0,Y 275.317,Z 376.319,A -85,B 0,C 180,E1 -17575.719,E2 -17575.719} C_VEL
LIN {X 0,Y 275.587,Z 375.265,A -85,B 0,C 180,E1 -17577.325,E2 -17577.325} C_VEL
LIN {X 0,Y 276.337,Z 372.167,A -85,B 0,C 180,E1 -17580.153,E2 -17580.153} C_VEL
LIN {X 0,Y 277.304,Z 367.823,A -85,B 0,C 180,E1 -17582.765,E2 -17582.765} C_VEL
LIN {X 0,Y 278.734,Z 361.673,A -85,B 0,C 180,E1 -17585.445,E2 -17585.445} C_VEL
LIN {X 0,Y 280.476,Z 354.28,A -85,B 0,C 180,E1 -17587.872,E2 -17587.872} C_VEL
LIN {X 0,Y 282.363,Z 345.996,A -85,B 0,C 180,E1 -17590.014,E2 -17590.014} C_VEL
LIN {X 0,Y 284.28,Z 336.922,A -85,B 0,C 180,E1 -17591.874,E2 -17591.874} C_VEL
LIN {X 0,Y 286.394,Z 326.078,A -85,B 0,C 180,E1 -17593.644,E2 -17593.644} C_VEL
LIN {X 0,Y 288.18,Z 315.508,A -85,B 0,C 180,E1 -17595.011,E2 -17595.011} C_VEL
LIN {X 0,Y 289.79,Z 303.917,A -85,B 0,C 180,E1 -17596.178,E2 -17596.178} C_VEL
LIN {X 0,Y 291.215,Z 290.631,A -85,B 0,C 180,E1 -17597.18,E2 -17597.18} C_VEL
LIN {X 0,Y 292.123,Z 278.138,A -85,B 0,C 180,E1 -17597.829,E2 -17597.829} C_VEL
LIN {X 0,Y 292.853,Z 262.29,A -85,B 0,C 180,E1 -17598.304,E2 -17598.304} C_VEL
LIN {X 0,Y 294.888,Z 203.074,A -85,B 0,C 180,E1 -17599.78,E2 -17599.78} C_VEL
LIN {X 0,Y 289.23,Z 189.363,A -85,B 0,C 180,E1 -17600.87,E2 -17600.87} C_VEL
LIN {X 0,Y 283.503,Z 177.483,A -85,B 0,C 180,E1 -17601.976,E2 -17601.976} C_VEL
LIN {X 0,Y 278.116,Z 167.01,A -85,B 0,C 180,E1 -17603.096,E2 -17603.096} C_VEL
LIN {X 0,Y 277.318,Z 163.944,A -85,B 0,C 180,E1 -17604.46,E2 -17604.46} C_VEL
LIN {X 0,Y 277.242,Z 163.949,A -85,B 0,C 180,E1 -17607.838,E2 -17607.838} C_VEL
LIN {X 0,Y 277.287,Z 163.945,A -85,B 0,C 180,E1 -17611.214,E2 -17611.214} C_VEL
LIN {X 0,Y 277.312,Z 163.946,A -85,B 0,C 180,E1 -17614.481,E2 -17614.481} C_VEL
LIN {X 0,Y 277.305,Z 163.94,A -85,B 0,C 180,E1 -17615.574,E2 -17615.574} C_VEL
LIN {X 0,Y 276.681,Z 164.023,A -85,B 0,C 180,E1 -17616.787,E2 -17616.787} C_VEL
LIN {X 0,Y 273.852,Z 164.377,A -85,B 0,C 180,E1 -17618.763,E2 -17618.763} C_VEL
LIN {X 0,Y 271.416,Z 164.68,A -85,B 0,C 180,E1 -17620.369,E2 -17620.369} C_VEL
LIN {X 0,Y 270.353,Z 164.808,A -85,B 0,C 180,E1 -17621.614,E2 -17621.614} C_VEL
LIN {X 0,Y 270.259,Z 164.816,A -85,B 0,C 180,E1 -17622.036,E2 -17622.036} C_VEL
LIN {X 0,Y 270.377,Z 164.807,A -85,B 0,C 180,E1 -17624.935,E2 -17624.935} C_VEL
LIN {X 0,Y 270.41,Z 164.8,A -85,B 0,C 180,E1 -17629.519,E2 -17629.519} C_VEL
LIN {X 0,Y 270.565,Z 164.776,A -85,B 0,C 180,E1 -17632.539,E2 -17632.539} C_VEL
LIN {X 0,Y 270.784,Z 164.751,A -85,B 0,C 180,E1 -17638.514,E2 -17638.514} C_VEL
LIN {X 0,Y 270.777,Z 164.74,A -85,B 0,C 180,E1 -17641.488,E2 -17641.488} C_VEL
LIN {X 0,Y 270.564,Z 164.775,A -85,B 0,C 180,E1 -17647.464,E2 -17647.464} C_VEL
LIN {X 0,Y 270.408,Z 164.785,A -85,B 0,C 180,E1 -17650.484,E2 -17650.484} C_VEL
LIN {X 0,Y 270.36,Z 164.802,A -85,B 0,C 180,E1 -17655.068,E2 -17655.068} C_VEL
LIN {X 0,Y 270.223,Z 164.822,A -85,B 0,C 180,E1 -17659.763,E2 -17659.763} C_VEL
LIN {X 0,Y 270.184,Z 164.828,A -85,B 0,C 180,E1 -17664.437,E2 -17664.437} C_VEL
LIN {X 0,Y 270.199,Z 164.828,A -85,B 0,C 180,E1 -17667.918,E2 -17667.918} C_VEL
LIN {X 0,Y 270.176,Z 164.823,A -85,B 0,C 180,E1 -17671.35,E2 -17671.35} C_VEL
LIN {X 0,Y 270.2,Z 164.82,A -85,B 0,C 180,E1 -17674.907,E2 -17674.907} C_VEL
LIN {X 0,Y 270.17,Z 164.827,A -85,B 0,C 180,E1 -17678.703,E2 -17678.703} C_VEL
LIN {X 0,Y 270.15,Z 164.837,A -85,B 0,C 180,E1 -17683.246,E2 -17683.246} C_VEL
LIN {X 0,Y 270.153,Z 164.839,A -85,B 0,C 180,E1 -17687.438,E2 -17687.438} C_VEL
LIN {X 0,Y 270.182,Z 164.957,A -85,B 0,C 180,E1 -17691.429,E2 -17691.429} C_VEL
LIN {X 0,Y 272.574,Z 173.609,A -85,B 0,C 180,E1 -17694.992,E2 -17694.992} C_VEL
LIN {X 0,Y 274.714,Z 182.975,A -85,B 0,C 180,E1 -17698.494,E2 -17698.494} C_VEL
LIN {X 0,Y 282.075,Z 199.457,A -85,B 0,C 180,E1 -17700.04,E2 -17700.04} C_VEL
LIN {X 0,Y 283.065,Z 202.436,A -85,B 0,C 180,E1 -17700.262,E2 -17700.262} C_VEL
LIN {X 0,Y 286.443,Z 222.478,A -85,B 0,C 180,E1 -17701.303,E2 -17701.303} C_VEL
LIN {X 0,Y 287.819,Z 233.989,A -85,B 0,C 180,E1 -17701.816,E2 -17701.816} C_VEL
LIN {X 0,Y 285.747,Z 292.785,A -85,B 0,C 180,E1 -17703.361,E2 -17703.361} C_VEL
LIN {X 0,Y 284.536,Z 306.613,A -85,B 0,C 180,E1 -17703.997,E2 -17703.997} C_VEL
LIN {X 0,Y 283.007,Z 318.838,A -85,B 0,C 180,E1 -17704.832,E2 -17704.832} C_VEL
LIN {X 0,Y 280.983,Z 331.422,A -85,B 0,C 180,E1 -17706.018,E2 -17706.018} C_VEL
LIN {X 0,Y 278.979,Z 342.656,A -85,B 0,C 180,E1 -17707.408,E2 -17707.408} C_VEL
LIN {X 0,Y 276.84,Z 352.816,A -85,B 0,C 180,E1 -17708.987,E2 -17708.987} C_VEL
LIN {X 0,Y 274.843,Z 362.183,A -85,B 0,C 180,E1 -17710.826,E2 -17710.826} C_VEL
LIN {X 0,Y 273.059,Z 370.26,A -85,B 0,C 180,E1 -17712.783,E2 -17712.783} C_VEL
LIN {X 0,Y 271.379,Z 377.613,A -85,B 0,C 180,E1 -17714.991,E2 -17714.991} C_VEL
LIN {X 0,Y 269.964,Z 383.528,A -85,B 0,C 180,E1 -17717.216,E2 -17717.216} C_VEL
LIN {X 0,Y 269.113,Z 388.21,A -85,B 0,C 180,E1 -17719.467,E2 -17719.467} C_VEL
LIN {X 0,Y 268.524,Z 391.797,A -85,B 0,C 180,E1 -17721.724,E2 -17721.724} C_VEL
LIN {X 0,Y 268.168,Z 395.082,A -85,B 0,C 180,E1 -17724.809,E2 -17724.809} C_VEL
LIN {X 0,Y 268.193,Z 396.379,A -85,B 0,C 180,E1 -17726.996,E2 -17726.996} C_VEL
LIN {X 0,Y 268.221,Z 396.763,A -85,B 0,C 180,E1 -17728.499,E2 -17728.499} C_VEL
LIN {X 0,Y 268.254,Z 396.758,A -85,B 0,C 180,E1 -17730,E2 -17730} C_VEL
LIN {X 0,Y 268.228,Z 396.353,A -85,B 0,C 180,E1 -17731.502,E2 -17731.502} C_VEL
LIN {X 0,Y 268.194,Z 395.501,A -85,B 0,C 180,E1 -17733.005,E2 -17733.005} C_VEL
LIN {X 0,Y 268.176,Z 393.534,A -85,B 0,C 180,E1 -17735.209,E2 -17735.209} C_VEL
LIN {X 0,Y 268.387,Z 390.448,A -85,B 0,C 180,E1 -17737.524,E2 -17737.524} C_VEL
LIN {X 0,Y 268.824,Z 386.352,A -85,B 0,C 180,E1 -17739.784,E2 -17739.784} C_VEL
LIN {X 0,Y 269.672,Z 380.046,A -85,B 0,C 180,E1 -17742.416,E2 -17742.416} C_VEL
LIN {X 0,Y 270.92,Z 373.183,A -85,B 0,C 180,E1 -17744.651,E2 -17744.651} C_VEL
LIN {X 0,Y 272.381,Z 365.085,A -85,B 0,C 180,E1 -17746.763,E2 -17746.763} C_VEL
LIN {X 0,Y 273.807,Z 355.765,A -85,B 0,C 180,E1 -17748.715,E2 -17748.715} C_VEL
LIN {X 0,Y 275.455,Z 346.082,A -85,B 0,C 180,E1 -17750.343,E2 -17750.343} C_VEL
LIN {X 0,Y 277.144,Z 335.505,A -85,B 0,C 180,E1 -17751.77,E2 -17751.77} C_VEL
LIN {X 0,Y 278.819,Z 323.79,A -85,B 0,C 180,E1 -17752.998,E2 -17752.998} C_VEL
LIN {X 0,Y 280.181,Z 311.625,A -85,B 0,C 180,E1 -17753.957,E2 -17753.957} C_VEL
LIN {X 0,Y 281.311,Z 298.425,A -85,B 0,C 180,E1 -17754.689,E2 -17754.689} C_VEL
LIN {X 0,Y 281.917,Z 285.457,A -85,B 0,C 180,E1 -17755.129,E2 -17755.129} C_VEL
LIN {X 0,Y 283.396,Z 231.043,A -85,B 0,C 180,E1 -17756.53,E2 -17756.53} C_VEL
LIN {X 0,Y 278.017,Z 194.582,A -85,B 0,C 180,E1 -17758.068,E2 -17758.068} C_VEL
LIN {X 0,Y 274.399,Z 184.133,A -85,B 0,C 180,E1 -17758.76,E2 -17758.76} C_VEL
LIN {X 0,Y 272.128,Z 173.138,A -85,B 0,C 180,E1 -17762.514,E2 -17762.514} C_VEL
LIN {X 0,Y 270.263,Z 164.817,A -85,B 0,C 180,E1 -17765.581,E2 -17765.581} C_VEL
LIN {X 0,Y 270.172,Z 164.827,A -85,B 0,C 180,E1 -17768.702,E2 -17768.702} C_VEL
LIN {X 0,Y 270.153,Z 164.83,A -85,B 0,C 180,E1 -17773.245,E2 -17773.245} C_VEL
LIN {X 0,Y 270.156,Z 164.835,A -85,B 0,C 180,E1 -17777.437,E2 -17777.437} C_VEL
LIN {X 0,Y 270.212,Z 164.829,A -85,B 0,C 180,E1 -17781.374,E2 -17781.374} C_VEL
LIN {X 0,Y 270.204,Z 164.831,A -85,B 0,C 180,E1 -17785.094,E2 -17785.094} C_VEL
LIN {X 0,Y 270.189,Z 164.831,A -85,B 0,C 180,E1 -17789.136,E2 -17789.136} C_VEL
LIN {X 0,Y 270.228,Z 164.823,A -85,B 0,C 180,E1 -17792.162,E2 -17792.162} C_VEL
LIN {X 0,Y 270.232,Z 164.822,A -85,B 0,C 180,E1 -17795.542,E2 -17795.542} C_VEL
LIN {X 0,Y 270.226,Z 164.823,A -85,B 0,C 180,E1 -17800.238,E2 -17800.238} C_VEL
LIN {X 0,Y 270.343,Z 164.809,A -85,B 0,C 180,E1 -17804.931,E2 -17804.931} C_VEL
LIN {X 0,Y 270.413,Z 164.795,A -85,B 0,C 180,E1 -17809.517,E2 -17809.517} C_VEL
LIN {X 0,Y 270.566,Z 164.771,A -85,B 0,C 180,E1 -17812.536,E2 -17812.536} C_VEL
LIN {X 0,Y 270.774,Z 164.756,A -85,B 0,C 180,E1 -17818.511,E2 -17818.511} C_VEL
LIN {X 0,Y 270.773,Z 164.748,A -85,B 0,C 180,E1 -17821.486,E2 -17821.486} C_VEL
LIN {X 0,Y 270.565,Z 164.778,A -85,B 0,C 180,E1 -17827.461,E2 -17827.461} C_VEL
LIN {X 0,Y 270.388,Z 164.803,A -85,B 0,C 180,E1 -17830.482,E2 -17830.482} C_VEL
LIN {X 0,Y 270.339,Z 164.796,A -85,B 0,C 180,E1 -17835.067,E2 -17835.067} C_VEL
LIN {X 0,Y 270.22,Z 164.824,A -85,B 0,C 180,E1 -17839.76,E2 -17839.76} C_VEL
LIN {X 0,Y 270.182,Z 164.824,A -85,B 0,C 180,E1 -17844.434,E2 -17844.434} C_VEL
LIN {X 0,Y 270.183,Z 164.818,A -85,B 0,C 180,E1 -17847.917,E2 -17847.917} C_VEL
LIN {X 0,Y 270.168,Z 164.83,A -85,B 0,C 180,E1 -17851.349,E2 -17851.349} C_VEL
LIN {X 0,Y 270.196,Z 164.826,A -85,B 0,C 180,E1 -17854.905,E2 -17854.905} C_VEL
LIN {X 0,Y 270.165,Z 164.82,A -85,B 0,C 180,E1 -17858.701,E2 -17858.701} C_VEL
LIN {X 0,Y 270.145,Z 164.837,A -85,B 0,C 180,E1 -17863.244,E2 -17863.244} C_VEL
LIN {X 0,Y 270.147,Z 164.828,A -85,B 0,C 180,E1 -17867.436,E2 -17867.436} C_VEL
LIN {X 0,Y 270.203,Z 164.829,A -85,B 0,C 180,E1 -17871.373,E2 -17871.373} C_VEL
LIN {X 0,Y 270.193,Z 164.824,A -85,B 0,C 180,E1 -17875.093,E2 -17875.093} C_VEL
LIN {X 0,Y 270.179,Z 164.83,A -85,B 0,C 180,E1 -17879.135,E2 -17879.135} C_VEL
LIN {X 0,Y 270.194,Z 164.824,A -85,B 0,C 180,E1 -17882.171,E2 -17882.171} C_VEL
LIN {X 0,Y 270.176,Z 164.826,A -85,B 0,C 180,E1 -17885.563,E2 -17885.563} C_VEL
LIN {X 0,Y 270.214,Z 164.828,A -85,B 0,C 180,E1 -17890.237,E2 -17890.237} C_VEL
LIN {X 0,Y 270.331,Z 164.809,A -85,B 0,C 180,E1 -17894.931,E2 -17894.931} C_VEL
LIN {X 0,Y 270.38,Z 164.803,A -85,B 0,C 180,E1 -17899.516,E2 -17899.516} C_VEL
LIN {X 0,Y 270.57,Z 164.981,A -85,B 0,C 180,E1 -17902.444,E2 -17902.444} C_VEL
LIN {X 0,Y 270.887,Z 166.359,A -85,B 0,C 180,E1 -17902.976,E2 -17902.976} C_VEL
LIN {X 0,Y 280.928,Z 190.979,A -85,B 0,C 180,E1 -17904.702,E2 -17904.702} C_VEL
LIN {X 0,Y 284.266,Z 200.907,A -85,B 0,C 180,E1 -17905.291,E2 -17905.291} C_VEL
LIN {X 0,Y 281.939,Z 274.052,A -85,B 0,C 180,E1 -17907.188,E2 -17907.188} C_VEL
LIN {X 0,Y 281.087,Z 287.348,A -85,B 0,C 180,E1 -17907.819,E2 -17907.819} C_VEL
LIN {X 0,Y 280.016,Z 300.287,A -85,B 0,C 180,E1 -17908.741,E2 -17908.741} C_VEL
LIN {X 0,Y 278.573,Z 313.057,A -85,B 0,C 180,E1 -17910,E2 -17910} C_VEL
LIN {X 0,Y 276.956,Z 324.473,A -85,B 0,C 180,E1 -17911.454,E2 -17911.454} C_VEL
LIN {X 0,Y 275.271,Z 334.849,A -85,B 0,C 180,E1 -17913.137,E2 -17913.137} C_VEL
LIN {X 0,Y 273.591,Z 344.764,A -85,B 0,C 180,E1 -17915.158,E2 -17915.158} C_VEL
LIN {X 0,Y 272.201,Z 352.25,A -85,B 0,C 180,E1 -17917.044,E2 -17917.044} C_VEL
LIN {X 0,Y 271.035,Z 358.45,A -85,B 0,C 180,E1 -17918.95,E2 -17918.95} C_VEL
LIN {X 0,Y 269.975,Z 364.51,A -85,B 0,C 180,E1 -17921.258,E2 -17921.258} C_VEL
LIN {X 0,Y 269.144,Z 369.259,A -85,B 0,C 180,E1 -17923.592,E2 -17923.592} C_VEL
LIN {X 0,Y 268.574,Z 372.842,A -85,B 0,C 180,E1 -17925.948,E2 -17925.948} C_VEL
LIN {X 0,Y 268.159,Z 375.358,A -85,B 0,C 180,E1 -17928.33,E2 -17928.33} C_VEL
LIN {X 0,Y 268.024,Z 376.446,A -85,B 0,C 180,E1 -17929.93,E2 -17929.93} C_VEL
LIN {X 0,Y 267.965,Z 377.111,A -85,B 0,C 180,E1 -17931.542,E2 -17931.542} C_VEL
LIN {X 0,Y 268.026,Z 377.28,A -85,B 0,C 180,E1 -17933.405,E2 -17933.405} C_VEL
LIN {X 0,Y 268.339,Z 376.295,A -85,B 0,C 180,E1 -17936.439,E2 -17936.439} C_VEL
LIN {X 0,Y 268.653,Z 375.048,A -85,B 0,C 180,E1 -17938.091,E2 -17938.091} C_VEL
LIN {X 0,Y 269.367,Z 372.238,A -85,B 0,C 180,E1 -17940.574,E2 -17940.574} C_VEL
LIN {X 0,Y 270.353,Z 368.143,A -85,B 0,C 180,E1 -17943.087,E2 -17943.087} C_VEL
LIN {X 0,Y 271.724,Z 362.653,A -85,B 0,C 180,E1 -17945.588,E2 -17945.588} C_VEL
LIN {X 0,Y 273.497,Z 355.456,A -85,B 0,C 180,E1 -17948.077,E2 -17948.077} C_VEL
LIN {X 0,Y 275.38,Z 347.702,A -85,B 0,C 180,E1 -17950.187,E2 -17950.187} C_VEL
LIN {X 0,Y 277.438,Z 338.632,A -85,B 0,C 180,E1 -17952.167,E2 -17952.167} C_VEL
LIN {X 0,Y 279.588,Z 328.099,A -85,B 0,C 180,E1 -17953.98,E2 -17953.98} C_VEL
LIN {X 0,Y 281.504,Z 317.537,A -85,B 0,C 180,E1 -17955.423,E2 -17955.423} C_VEL
LIN {X 0,Y 283.268,Z 306.06,A -85,B 0,C 180,E1 -17956.657,E2 -17956.657} C_VEL
LIN {X 0,Y 284.684,Z 293.79,A -85,B 0,C 180,E1 -17957.652,E2 -17957.652} C_VEL
LIN {X 0,Y 285.753,Z 280.314,A -85,B 0,C 180,E1 -17958.429,E2 -17958.429} C_VEL
LIN {X 0,Y 286.53,Z 267.547,A -85,B 0,C 180,E1 -17958.862,E2 -17958.862} C_VEL
LIN {X 0,Y 288.67,Z 204.613,A -85,B 0,C 180,E1 -17960.482,E2 -17960.482} C_VEL
LIN {X 0,Y 282.544,Z 189.996,A -85,B 0,C 180,E1 -17961.715,E2 -17961.715} C_VEL
LIN {X 0,Y 276.214,Z 177.355,A -85,B 0,C 180,E1 -17962.995,E2 -17962.995} C_VEL
LIN {X 0,Y 272.034,Z 169.754,A -85,B 0,C 180,E1 -17963.867,E2 -17963.867} C_VEL
LIN {X 0,Y 270.896,Z 167.331,A -85,B 0,C 180,E1 -17964.166,E2 -17964.166} C_VEL
LIN {X 0,Y 270.241,Z 164.828,A -85,B 0,C 180,E1 -17965.275,E2 -17965.275} C_VEL
LIN {X 0,Y 270.226,Z 164.821,A -85,B 0,C 180,E1 -17970.388,E2 -17970.388} C_VEL
LIN {X 0,Y 270.262,Z 164.822,A -85,B 0,C 180,E1 -17973.765,E2 -17973.765} C_VEL
LIN {X 0,Y 270.231,Z 164.827,A -85,B 0,C 180,E1 -17977.04,E2 -17977.04} C_VEL
LIN {X 0,Y 270.296,Z 164.816,A -85,B 0,C 180,E1 -17980.245,E2 -17980.245} C_VEL
LIN {X 0,Y 270.259,Z 164.816,A -85,B 0,C 180,E1 -17982.036,E2 -17982.036} C_VEL
LIN {X 0,Y 269.576,Z 164.901,A -85,B 0,C 180,E1 -17983.28,E2 -17983.28} C_VEL
LIN {X 0,Y 266.747,Z 165.256,A -85,B 0,C 180,E1 -17985.31,E2 -17985.31} C_VEL
LIN {X 0,Y 264.379,Z 165.547,A -85,B 0,C 180,E1 -17986.96,E2 -17986.96} C_VEL
LIN {X 0,Y 263.389,Z 165.674,A -85,B 0,C 180,E1 -17988.238,E2 -17988.238} C_VEL
LIN {X 0,Y 263.322,Z 165.679,A -85,B 0,C 180,E1 -17988.671,E2 -17988.671} C_VEL
LIN {X 0,Y 263.528,Z 165.651,A -85,B 0,C 180,E1 -17992.338,E2 -17992.338} C_VEL
LIN {X 0,Y 263.748,Z 165.628,A -85,B 0,C 180,E1 -17998.474,E2 -17998.474} C_VEL
LIN {X 0,Y 263.74,Z 165.617,A -85,B 0,C 180,E1 -18001.528,E2 -18001.528} C_VEL
LIN {X 0,Y 263.528,Z 165.652,A -85,B 0,C 180,E1 -18007.664,E2 -18007.664} C_VEL
LIN {X 0,Y 263.347,Z 165.663,A -85,B 0,C 180,E1 -18010.768,E2 -18010.768} C_VEL
LIN {X 0,Y 263.304,Z 165.676,A -85,B 0,C 180,E1 -18015.482,E2 -18015.482} C_VEL
LIN {X 0,Y 263.21,Z 165.692,A -85,B 0,C 180,E1 -18020.312,E2 -18020.312} C_VEL
LIN {X 0,Y 263.128,Z 165.7,A -85,B 0,C 180,E1 -18025.301,E2 -18025.301} C_VEL
LIN {X 0,Y 263.135,Z 165.708,A -85,B 0,C 180,E1 -18028.736,E2 -18028.736} C_VEL
LIN {X 0,Y 263.131,Z 165.708,A -85,B 0,C 180,E1 -18032.29,E2 -18032.29} C_VEL
LIN {X 0,Y 263.157,Z 165.706,A -85,B 0,C 180,E1 -18035.984,E2 -18035.984} C_VEL
LIN {X 0,Y 263.075,Z 165.718,A -85,B 0,C 180,E1 -18039.879,E2 -18039.879} C_VEL
LIN {X 0,Y 263.079,Z 165.715,A -85,B 0,C 180,E1 -18043.995,E2 -18043.995} C_VEL
LIN {X 0,Y 263.078,Z 165.722,A -85,B 0,C 180,E1 -18048.098,E2 -18048.098} C_VEL
LIN {X 0,Y 263.103,Z 165.826,A -85,B 0,C 180,E1 -18050.469,E2 -18050.469} C_VEL
LIN {X 0,Y 265.362,Z 173.905,A -85,B 0,C 180,E1 -18053.956,E2 -18053.956} C_VEL
LIN {X 0,Y 267.495,Z 182.694,A -85,B 0,C 180,E1 -18057.392,E2 -18057.392} C_VEL
LIN {X 0,Y 274.868,Z 198.528,A -85,B 0,C 180,E1 -18059.024,E2 -18059.024} C_VEL
LIN {X 0,Y 277.303,Z 204.757,A -85,B 0,C 180,E1 -18059.564,E2 -18059.564} C_VEL
LIN {X 0,Y 280.765,Z 226.219,A -85,B 0,C 180,E1 -18060.698,E2 -18060.698} C_VEL
LIN {X 0,Y 281.749,Z 234.595,A -85,B 0,C 180,E1 -18061.082,E2 -18061.082} C_VEL
LIN {X 0,Y 279.603,Z 292.508,A -85,B 0,C 180,E1 -18062.638,E2 -18062.638} C_VEL
LIN {X 0,Y 278.369,Z 306.143,A -85,B 0,C 180,E1 -18063.275,E2 -18063.275} C_VEL
LIN {X 0,Y 276.762,Z 318.412,A -85,B 0,C 180,E1 -18064.122,E2 -18064.122} C_VEL
LIN {X 0,Y 274.811,Z 330.23,A -85,B 0,C 180,E1 -18065.243,E2 -18065.243} C_VEL
LIN {X 0,Y 272.69,Z 341.615,A -85,B 0,C 180,E1 -18066.656,E2 -18066.656} C_VEL
LIN {X 0,Y 270.459,Z 351.935,A -85,B 0,C 180,E1 -18068.267,E2 -18068.267} C_VEL
LIN {X 0,Y 268.365,Z 361.228,A -85,B 0,C 180,E1 -18070.096,E2 -18070.096} C_VEL
LIN {X 0,Y 266.289,Z 370.268,A -85,B 0,C 180,E1 -18072.332,E2 -18072.332} C_VEL
LIN {X 0,Y 264.526,Z 377.575,A -85,B 0,C 180,E1 -18074.593,E2 -18074.593} C_VEL
LIN {X 0,Y 263.028,Z 383.445,A -85,B 0,C 180,E1 -18076.873,E2 -18076.873} C_VEL
LIN {X 0,Y 262.086,Z 388.088,A -85,B 0,C 180,E1 -18079.181,E2 -18079.181} C_VEL
LIN {X 0,Y 261.467,Z 391.639,A -85,B 0,C 180,E1 -18081.499,E2 -18081.499} C_VEL
LIN {X 0,Y 261.151,Z 394.189,A -85,B 0,C 180,E1 -18083.821,E2 -18083.821} C_VEL
LIN {X 0,Y 261.07,Z 395.381,A -85,B 0,C 180,E1 -18085.368,E2 -18085.368} C_VEL
LIN {X 0,Y 261.104,Z 396.141,A -85,B 0,C 180,E1 -18086.914,E2 -18086.914} C_VEL
LIN {X 0,Y 261.146,Z 396.511,A -85,B 0,C 180,E1 -18088.458,E2 -18088.458} C_VEL
LIN {X 0,Y 261.178,Z 396.491,A -85,B 0,C 180,E1 -18090,E2 -18090} C_VEL
LIN {X 0,Y 261.153,Z 396.063,A -85,B 0,C 180,E1 -18091.542,E2 -18091.542} C_VEL
LIN {X 0,Y 261.105,Z 395.191,A -85,B 0,C 180,E1 -18093.086,E2 -18093.086} C_VEL
LIN {X 0,Y 261.088,Z 393.434,A -85,B 0,C 180,E1 -18095.136,E2 -18095.136} C_VEL
LIN {X 0,Y 261.328,Z 390.074,A -85,B 0,C 180,E1 -18097.728,E2 -18097.728} C_VEL
LIN {X 0,Y 261.779,Z 385.942,A -85,B 0,C 180,E1 -18100.05,E2 -18100.05} C_VEL
LIN {X 0,Y 262.705,Z 379.6,A -85,B 0,C 180,E1 -18102.751,E2 -18102.751} C_VEL
LIN {X 0,Y 264.011,Z 372.691,A -85,B 0,C 180,E1 -18105.044,E2 -18105.044} C_VEL
LIN {X 0,Y 265.561,Z 364.135,A -85,B 0,C 180,E1 -18107.298,E2 -18107.298} C_VEL
LIN {X 0,Y 267.003,Z 355.12,A -85,B 0,C 180,E1 -18109.21,E2 -18109.21} C_VEL
LIN {X 0,Y 268.979,Z 344.175,A -85,B 0,C 180,E1 -18111.056,E2 -18111.056} C_VEL
LIN {X 0,Y 270.756,Z 333.118,A -85,B 0,C 180,E1 -18112.512,E2 -18112.512} C_VEL
LIN {X 0,Y 272.454,Z 320.735,A -85,B 0,C 180,E1 -18113.769,E2 -18113.769} C_VEL
LIN {X 0,Y 273.863,Z 309.042,A -85,B 0,C 180,E1 -18114.647,E2 -18114.647} C_VEL
LIN {X 0,Y 274.893,Z 296.524,A -85,B 0,C 180,E1 -18115.306,E2 -18115.306} C_VEL
LIN {X 0,Y 275.574,Z 279.368,A -85,B 0,C 180,E1 -18115.838,E2 -18115.838} C_VEL
LIN {X 0,Y 276.83,Z 231.479,A -85,B 0,C 180,E1 -18117.107,E2 -18117.107} C_VEL
LIN {X 0,Y 271.75,Z 196.649,A -85,B 0,C 180,E1 -18118.618,E2 -18118.618} C_VEL
LIN {X 0,Y 267.916,Z 186.214,A -85,B 0,C 180,E1 -18119.326,E2 -18119.326} C_VEL
LIN {X 0,Y 267.118,Z 183.817,A -85,B 0,C 180,E1 -18119.527,E2 -18119.527} C_VEL
LIN {X 0,Y 264.828,Z 172.829,A -85,B 0,C 180,E1 -18123.413,E2 -18123.413} C_VEL
LIN {X 0,Y 263.209,Z 165.697,A -85,B 0,C 180,E1 -18126.071,E2 -18126.071} C_VEL
LIN {X 0,Y 263.077,Z 165.718,A -85,B 0,C 180,E1 -18129.878,E2 -18129.878} C_VEL
LIN {X 0,Y 263.081,Z 165.714,A -85,B 0,C 180,E1 -18133.994,E2 -18133.994} C_VEL
LIN {X 0,Y 263.085,Z 165.714,A -85,B 0,C 180,E1 -18138.417,E2 -18138.417} C_VEL
LIN {X 0,Y 263.163,Z 165.704,A -85,B 0,C 180,E1 -18142.102,E2 -18142.102} C_VEL
LIN {X 0,Y 263.156,Z 165.705,A -85,B 0,C 180,E1 -18145.885,E2 -18145.885} C_VEL
LIN {X 0,Y 263.131,Z 165.708,A -85,B 0,C 180,E1 -18149.503,E2 -18149.503} C_VEL
LIN {X 0,Y 263.147,Z 165.708,A -85,B 0,C 180,E1 -18152.996,E2 -18152.996} C_VEL
LIN {X 0,Y 263.149,Z 165.706,A -85,B 0,C 180,E1 -18156.382,E2 -18156.382} C_VEL
LIN {X 0,Y 263.213,Z 165.695,A -85,B 0,C 180,E1 -18159.688,E2 -18159.688} C_VEL
LIN {X 0,Y 263.292,Z 165.69,A -85,B 0,C 180,E1 -18164.517,E2 -18164.517} C_VEL
LIN {X 0,Y 263.352,Z 165.675,A -85,B 0,C 180,E1 -18169.232,E2 -18169.232} C_VEL
LIN {X 0,Y 263.53,Z 165.645,A -85,B 0,C 180,E1 -18172.336,E2 -18172.336} C_VEL
LIN {X 0,Y 263.737,Z 165.632,A -85,B 0,C 180,E1 -18178.472,E2 -18178.472} C_VEL
LIN {X 0,Y 263.737,Z 165.625,A -85,B 0,C 180,E1 -18181.526,E2 -18181.526} C_VEL
LIN {X 0,Y 263.528,Z 165.656,A -85,B 0,C 180,E1 -18187.662,E2 -18187.662} C_VEL
LIN {X 0,Y 263.332,Z 165.68,A -85,B 0,C 180,E1 -18190.766,E2 -18190.766} C_VEL
LIN {X 0,Y 263.289,Z 165.673,A -85,B 0,C 180,E1 -18195.48,E2 -18195.48} C_VEL
LIN {X 0,Y 263.208,Z 165.697,A -85,B 0,C 180,E1 -18200.31,E2 -18200.31} C_VEL
LIN {X 0,Y 263.12,Z 165.704,A -85,B 0,C 180,E1 -18205.299,E2 -18205.299} C_VEL
LIN {X 0,Y 263.117,Z 165.698,A -85,B 0,C 180,E1 -18208.735,E2 -18208.735} C_VEL
LIN {X 0,Y 263.125,Z 165.707,A -85,B 0,C 180,E1 -18212.288,E2 -18212.288} C_VEL
LIN {X 0,Y 263.152,Z 165.698,A -85,B 0,C 180,E1 -18215.982,E2 -18215.982} C_VEL
LIN {X 0,Y 263.079,Z 165.71,A -85,B 0,C 180,E1 -18219.875,E2 -18219.875} C_VEL
LIN {X 0,Y 263.073,Z 165.714,A -85,B 0,C 180,E1 -18223.993,E2 -18223.993} C_VEL
LIN {X 0,Y 263.076,Z 165.708,A -85,B 0,C 180,E1 -18228.416,E2 -18228.416} C_VEL
LIN {X 0,Y 263.153,Z 165.706,A -85,B 0,C 180,E1 -18232.101,E2 -18232.101} C_VEL
LIN {X 0,Y 263.147,Z 165.702,A -85,B 0,C 180,E1 -18235.884,E2 -18235.884} C_VEL
LIN {X 0,Y 263.121,Z 165.708,A -85,B 0,C 180,E1 -18239.502,E2 -18239.502} C_VEL
LIN {X 0,Y 263.121,Z 165.71,A -85,B 0,C 180,E1 -18242.994,E2 -18242.994} C_VEL
LIN {X 0,Y 263.109,Z 165.705,A -85,B 0,C 180,E1 -18246.379,E2 -18246.379} C_VEL
LIN {X 0,Y 263.201,Z 165.699,A -85,B 0,C 180,E1 -18249.688,E2 -18249.688} C_VEL
LIN {X 0,Y 263.281,Z 165.69,A -85,B 0,C 180,E1 -18254.517,E2 -18254.517} C_VEL
LIN {X 0,Y 263.325,Z 165.681,A -85,B 0,C 180,E1 -18259.232,E2 -18259.232} C_VEL
LIN {X 0,Y 263.495,Z 165.765,A -85,B 0,C 180,E1 -18261.869,E2 -18261.869} C_VEL
LIN {X 0,Y 263.691,Z 166.637,A -85,B 0,C 180,E1 -18262.214,E2 -18262.214} C_VEL
LIN {X 0,Y 274.797,Z 193.571,A -85,B 0,C 180,E1 -18264.19,E2 -18264.19} C_VEL
LIN {X 0,Y 277.779,Z 202.316,A -85,B 0,C 180,E1 -18264.732,E2 -18264.732} C_VEL
LIN {X 0,Y 275.392,Z 274.152,A -85,B 0,C 180,E1 -18266.633,E2 -18266.633} C_VEL
LIN {X 0,Y 274.435,Z 287.872,A -85,B 0,C 180,E1 -18267.295,E2 -18267.295} C_VEL
LIN {X 0,Y 273.349,Z 300.836,A -85,B 0,C 180,E1 -18268.251,E2 -18268.251} C_VEL
LIN {X 0,Y 271.971,Z 312.727,A -85,B 0,C 180,E1 -18269.444,E2 -18269.444} C_VEL
LIN {X 0,Y 270.276,Z 324.262,A -85,B 0,C 180,E1 -18270.931,E2 -18270.931} C_VEL
LIN {X 0,Y 268.568,Z 334.597,A -85,B 0,C 180,E1 -18272.624,E2 -18272.624} C_VEL
LIN {X 0,Y 266.929,Z 343.89,A -85,B 0,C 180,E1 -18274.53,E2 -18274.53} C_VEL
LIN {X 0,Y 265.203,Z 352.961,A -85,B 0,C 180,E1 -18276.849,E2 -18276.849} C_VEL
LIN {X 0,Y 263.789,Z 360.168,A -85,B 0,C 180,E1 -18279.198,E2 -18279.198} C_VEL
LIN {X 0,Y 262.747,Z 365.901,A -85,B 0,C 180,E1 -18281.572,E2 -18281.572} C_VEL
LIN {X 0,Y 261.94,Z 370.388,A -85,B 0,C 180,E1 -18283.973,E2 -18283.973} C_VEL
LIN {X 0,Y 261.553,Z 372.763,A -85,B 0,C 180,E1 -18285.587,E2 -18285.587} C_VEL
LIN {X 0,Y 261.219,Z 374.622,A -85,B 0,C 180,E1 -18287.214,E2 -18287.214} C_VEL
LIN {X 0,Y 260.967,Z 376.476,A -85,B 0,C 180,E1 -18289.517,E2 -18289.517} C_VEL
LIN {X 0,Y 260.875,Z 377.478,A -85,B 0,C 180,E1 -18292.158,E2 -18292.158} C_VEL
LIN {X 0,Y 260.965,Z 377.515,A -85,B 0,C 180,E1 -18293.826,E2 -18293.826} C_VEL
LIN {X 0,Y 261.123,Z 377.113,A -85,B 0,C 180,E1 -18295.508,E2 -18295.508} C_VEL
LIN {X 0,Y 261.43,Z 375.983,A -85,B 0,C 180,E1 -18297.488,E2 -18297.488} C_VEL
LIN {X 0,Y 261.773,Z 374.792,A -85,B 0,C 180,E1 -18298.898,E2 -18298.898} C_VEL
LIN {X 0,Y 262.432,Z 372.308,A -85,B 0,C 180,E1 -18301.025,E2 -18301.025} C_VEL
LIN {X 0,Y 263.298,Z 368.93,A -85,B 0,C 180,E1 -18303.174,E2 -18303.174} C_VEL
LIN {X 0,Y 264.714,Z 363.587,A -85,B 0,C 180,E1 -18305.738,E2 -18305.738} C_VEL
LIN {X 0,Y 266.466,Z 356.899,A -85,B 0,C 180,E1 -18308.206,E2 -18308.206} C_VEL
LIN {X 0,Y 268.355,Z 349.603,A -85,B 0,C 180,E1 -18310.316,E2 -18310.316} C_VEL
LIN {X 0,Y 270.595,Z 340.235,A -85,B 0,C 180,E1 -18312.476,E2 -18312.476} C_VEL
LIN {X 0,Y 272.8,Z 330.131,A -85,B 0,C 180,E1 -18314.331,E2 -18314.331} C_VEL
LIN {X 0,Y 274.662,Z 320.355,A -85,B 0,C 180,E1 -18315.763,E2 -18315.763} C_VEL
LIN {X 0,Y 276.71,Z 308.576,A -85,B 0,C 180,E1 -18317.107,E2 -18317.107} C_VEL
LIN {X 0,Y 278.213,Z 296.536,A -85,B 0,C 180,E1 -18318.177,E2 -18318.177} C_VEL
LIN {X 0,Y 279.389,Z 283.669,A -85,B 0,C 180,E1 -18318.994,E2 -18318.994} C_VEL
LIN {X 0,Y 280.295,Z 270.422,A -85,B 0,C 180,E1 -18319.513,E2 -18319.513} C_VEL
LIN {X 0,Y 282.649,Z 206.63,A -85,B 0,C 180,E1 -18321.186,E2 -18321.186} C_VEL
LIN {X 0,Y 276.916,Z 192.926,A -85,B 0,C 180,E1 -18322.39,E2 -18322.39} C_VEL
LIN {X 0,Y 269.503,Z 178.182,A -85,B 0,C 180,E1 -18323.972,E2 -18323.972} C_VEL
LIN {X 0,Y 265.02,Z 170.375,A -85,B 0,C 180,E1 -18324.952,E2 -18324.952} C_VEL
LIN {X 0,Y 263.733,Z 167.676,A -85,B 0,C 180,E1 -18325.303,E2 -18325.303} C_VEL
LIN {X 0,Y 263.182,Z 165.702,A -85,B 0,C 180,E1 -18326.267,E2 -18326.267} C_VEL
LIN {X 0,Y 263.148,Z 165.707,A -85,B 0,C 180,E1 -18329.508,E2 -18329.508} C_VEL
LIN {X 0,Y 263.191,Z 165.699,A -85,B 0,C 180,E1 -18333.004,E2 -18333.004} C_VEL
LIN {X 0,Y 263.182,Z 165.701,A -85,B 0,C 180,E1 -18336.388,E2 -18336.388} C_VEL
LIN {X 0,Y 263.261,Z 165.689,A -85,B 0,C 180,E1 -18339.695,E2 -18339.695} C_VEL
LIN {X 0,Y 263.323,Z 165.685,A -85,B 0,C 180,E1 -18344.522,E2 -18344.522} C_VEL
LIN {X 0,Y 263.322,Z 165.679,A -85,B 0,C 180,E1 -18348.671,E2 -18348.671} C_VEL
LIN {X 0,Y 262.679,Z 165.764,A -85,B 0,C 180,E1 -18349.949,E2 -18349.949} C_VEL
LIN {X 0,Y 259.811,Z 166.121,A -85,B 0,C 180,E1 -18352.032,E2 -18352.032} C_VEL
LIN {X 0,Y 257.387,Z 166.421,A -85,B 0,C 180,E1 -18353.727,E2 -18353.727} C_VEL
LIN {X 0,Y 256.39,Z 166.535,A -85,B 0,C 180,E1 -18355.041,E2 -18355.041} C_VEL
LIN {X 0,Y 256.332,Z 166.539,A -85,B 0,C 180,E1 -18355.486,E2 -18355.486} C_VEL
LIN {X 0,Y 256.711,Z 166.505,A -85,B 0,C 180,E1 -18358.433,E2 -18358.433} C_VEL
LIN {X 0,Y 256.702,Z 166.493,A -85,B 0,C 180,E1 -18361.57,E2 -18361.57} C_VEL
LIN {X 0,Y 256.457,Z 166.522,A -85,B 0,C 180,E1 -18366.294,E2 -18366.294} C_VEL
LIN {X 0,Y 256.428,Z 166.537,A -85,B 0,C 180,E1 -18369.466,E2 -18369.466} C_VEL
LIN {X 0,Y 256.226,Z 166.566,A -85,B 0,C 180,E1 -18374.293,E2 -18374.293} C_VEL
LIN {X 0,Y 256.161,Z 166.568,A -85,B 0,C 180,E1 -18377.567,E2 -18377.567} C_VEL
LIN {X 0,Y 256.121,Z 166.569,A -85,B 0,C 180,E1 -18381.098,E2 -18381.098} C_VEL
LIN {X 0,Y 256.087,Z 166.579,A -85,B 0,C 180,E1 -18385.09,E2 -18385.09} C_VEL
LIN {X 0,Y 256.092,Z 166.585,A -85,B 0,C 180,E1 -18388.576,E2 -18388.576} C_VEL
LIN {X 0,Y 256.077,Z 166.582,A -85,B 0,C 180,E1 -18391.702,E2 -18391.702} C_VEL
LIN {X 0,Y 256.08,Z 166.58,A -85,B 0,C 180,E1 -18395.195,E2 -18395.195} C_VEL
LIN {X 0,Y 256.044,Z 166.59,A -85,B 0,C 180,E1 -18399.148,E2 -18399.148} C_VEL
LIN {X 0,Y 256.024,Z 166.597,A -85,B 0,C 180,E1 -18403.337,E2 -18403.337} C_VEL
LIN {X 0,Y 256.033,Z 166.6,A -85,B 0,C 180,E1 -18407.83,E2 -18407.83} C_VEL
LIN {X 0,Y 256.022,Z 166.601,A -85,B 0,C 180,E1 -18409.38,E2 -18409.38} C_VEL
LIN {X 0,Y 258.469,Z 175.155,A -85,B 0,C 180,E1 -18413.259,E2 -18413.259} C_VEL
LIN {X 0,Y 260.221,Z 182.334,A -85,B 0,C 180,E1 -18416.19,E2 -18416.19} C_VEL
LIN {X 0,Y 267.077,Z 196.541,A -85,B 0,C 180,E1 -18417.798,E2 -18417.798} C_VEL
LIN {X 0,Y 271.598,Z 207.173,A -85,B 0,C 180,E1 -18418.833,E2 -18418.833} C_VEL
LIN {X 0,Y 274.933,Z 228.46,A -85,B 0,C 180,E1 -18419.995,E2 -18419.995} C_VEL
LIN {X 0,Y 275.737,Z 235.166,A -85,B 0,C 180,E1 -18420.316,E2 -18420.316} C_VEL
LIN {X 0,Y 273.545,Z 292.118,A -85,B 0,C 180,E1 -18421.877,E2 -18421.877} C_VEL
LIN {X 0,Y 272.232,Z 305.768,A -85,B 0,C 180,E1 -18422.518,E2 -18422.518} C_VEL
LIN {X 0,Y 270.564,Z 318.068,A -85,B 0,C 180,E1 -18423.38,E2 -18423.38} C_VEL
LIN {X 0,Y 268.72,Z 329.115,A -85,B 0,C 180,E1 -18424.435,E2 -18424.435} C_VEL
LIN {X 0,Y 266.475,Z 340.655,A -85,B 0,C 180,E1 -18425.871,E2 -18425.871} C_VEL
LIN {X 0,Y 264.132,Z 351.08,A -85,B 0,C 180,E1 -18427.512,E2 -18427.512} C_VEL
LIN {X 0,Y 262.058,Z 359.626,A -85,B 0,C 180,E1 -18429.186,E2 -18429.186} C_VEL
LIN {X 0,Y 260.217,Z 367.528,A -85,B 0,C 180,E1 -18431.089,E2 -18431.089} C_VEL
LIN {X 0,Y 258.264,Z 375.283,A -85,B 0,C 180,E1 -18433.398,E2 -18433.398} C_VEL
LIN {X 0,Y 256.568,Z 381.535,A -85,B 0,C 180,E1 -18435.728,E2 -18435.728} C_VEL
LIN {X 0,Y 255.377,Z 386.525,A -85,B 0,C 180,E1 -18438.089,E2 -18438.089} C_VEL
LIN {X 0,Y 254.618,Z 390.397,A -85,B 0,C 180,E1 -18440.467,E2 -18440.467} C_VEL
LIN {X 0,Y 254.061,Z 394.002,A -85,B 0,C 180,E1 -18443.647,E2 -18443.647} C_VEL
LIN {X 0,Y 253.977,Z 395.16,A -85,B 0,C 180,E1 -18445.238,E2 -18445.238} C_VEL
LIN {X 0,Y 254,Z 395.904,A -85,B 0,C 180,E1 -18446.828,E2 -18446.828} C_VEL
LIN {X 0,Y 254.073,Z 396.26,A -85,B 0,C 180,E1 -18448.415,E2 -18448.415} C_VEL
LIN {X 0,Y 254.103,Z 396.224,A -85,B 0,C 180,E1 -18450,E2 -18450} C_VEL
LIN {X 0,Y 254.079,Z 395.764,A -85,B 0,C 180,E1 -18451.585,E2 -18451.585} C_VEL
LIN {X 0,Y 254.019,Z 394.873,A -85,B 0,C 180,E1 -18453.172,E2 -18453.172} C_VEL
LIN {X 0,Y 253.987,Z 393.341,A -85,B 0,C 180,E1 -18455.021,E2 -18455.021} C_VEL
LIN {X 0,Y 254.265,Z 389.684,A -85,B 0,C 180,E1 -18457.944,E2 -18457.944} C_VEL
LIN {X 0,Y 254.752,Z 385.511,A -85,B 0,C 180,E1 -18460.331,E2 -18460.331} C_VEL
LIN {X 0,Y 255.724,Z 379.122,A -85,B 0,C 180,E1 -18463.105,E2 -18463.105} C_VEL
LIN {X 0,Y 257.088,Z 372.164,A -85,B 0,C 180,E1 -18465.459,E2 -18465.459} C_VEL
LIN {X 0,Y 258.661,Z 363.92,A -85,B 0,C 180,E1 -18467.675,E2 -18467.675} C_VEL
LIN {X 0,Y 260.262,Z 354.438,A -85,B 0,C 180,E1 -18469.728,E2 -18469.728} C_VEL
LIN {X 0,Y 262.113,Z 344.592,A -85,B 0,C 180,E1 -18471.428,E2 -18471.428} C_VEL
LIN {X 0,Y 263.929,Z 333.761,A -85,B 0,C 180,E1 -18472.92,E2 -18472.92} C_VEL
LIN {X 0,Y 265.698,Z 321.611,A -85,B 0,C 180,E1 -18474.205,E2 -18474.205} C_VEL
LIN {X 0,Y 267.263,Z 308.962,A -85,B 0,C 180,E1 -18475.194,E2 -18475.194} C_VEL
LIN {X 0,Y 268.319,Z 296.571,A -85,B 0,C 180,E1 -18475.867,E2 -18475.867} C_VEL
LIN {X 0,Y 269.041,Z 279.653,A -85,B 0,C 180,E1 -18476.407,E2 -18476.407} C_VEL
LIN {X 0,Y 270.352,Z 232.389,A -85,B 0,C 180,E1 -18477.688,E2 -18477.688} C_VEL
LIN {X 0,Y 265.605,Z 199.301,A -85,B 0,C 180,E1 -18479.167,E2 -18479.167} C_VEL
LIN {X 0,Y 262.556,Z 190.511,A -85,B 0,C 180,E1 -18479.763,E2 -18479.763} C_VEL
LIN {X 0,Y 259.886,Z 183.633,A -85,B 0,C 180,E1 -18480.287,E2 -18480.287} C_VEL
LIN {X 0,Y 257.738,Z 173.531,A -85,B 0,C 180,E1 -18483.987,E2 -18483.987} C_VEL
LIN {X 0,Y 256.113,Z 166.584,A -85,B 0,C 180,E1 -18486.706,E2 -18486.706} C_VEL
LIN {X 0,Y 256.013,Z 166.593,A -85,B 0,C 180,E1 -18491.212,E2 -18491.212} C_VEL
LIN {X 0,Y 256.022,Z 166.595,A -85,B 0,C 180,E1 -18495.539,E2 -18495.539} C_VEL
LIN {X 0,Y 256.023,Z 166.595,A -85,B 0,C 180,E1 -18498.789,E2 -18498.789} C_VEL
LIN {X 0,Y 256.133,Z 166.583,A -85,B 0,C 180,E1 -18502.866,E2 -18502.866} C_VEL
LIN {X 0,Y 256.071,Z 166.589,A -85,B 0,C 180,E1 -18506.706,E2 -18506.706} C_VEL
LIN {X 0,Y 256.06,Z 166.589,A -85,B 0,C 180,E1 -18510.392,E2 -18510.392} C_VEL
LIN {X 0,Y 256.138,Z 166.581,A -85,B 0,C 180,E1 -18514.888,E2 -18514.888} C_VEL
LIN {X 0,Y 256.129,Z 166.579,A -85,B 0,C 180,E1 -18519.1,E2 -18519.1} C_VEL
LIN {X 0,Y 256.217,Z 166.569,A -85,B 0,C 180,E1 -18524.079,E2 -18524.079} C_VEL
LIN {X 0,Y 256.292,Z 166.555,A -85,B 0,C 180,E1 -18528.932,E2 -18528.932} C_VEL
LIN {X 0,Y 256.473,Z 166.522,A -85,B 0,C 180,E1 -18532.124,E2 -18532.124} C_VEL
LIN {X 0,Y 256.455,Z 166.539,A -85,B 0,C 180,E1 -18536.857,E2 -18536.857} C_VEL
LIN {X 0,Y 256.7,Z 166.509,A -85,B 0,C 180,E1 -18538.43,E2 -18538.43} C_VEL
LIN {X 0,Y 256.699,Z 166.501,A -85,B 0,C 180,E1 -18541.568,E2 -18541.568} C_VEL
LIN {X 0,Y 256.449,Z 166.534,A -85,B 0,C 180,E1 -18546.574,E2 -18546.574} C_VEL
LIN {X 0,Y 256.404,Z 166.545,A -85,B 0,C 180,E1 -18549.464,E2 -18549.464} C_VEL
LIN {X 0,Y 256.202,Z 166.556,A -85,B 0,C 180,E1 -18554.292,E2 -18554.292} C_VEL
LIN {X 0,Y 256.148,Z 166.566,A -85,B 0,C 180,E1 -18557.565,E2 -18557.565} C_VEL
LIN {X 0,Y 256.119,Z 166.58,A -85,B 0,C 180,E1 -18561.095,E2 -18561.095} C_VEL
LIN {X 0,Y 256.082,Z 166.581,A -85,B 0,C 180,E1 -18565.086,E2 -18565.086} C_VEL
LIN {X 0,Y 256.075,Z 166.574,A -85,B 0,C 180,E1 -18568.568,E2 -18568.568} C_VEL
LIN {X 0,Y 256.069,Z 166.589,A -85,B 0,C 180,E1 -18571.698,E2 -18571.698} C_VEL
LIN {X 0,Y 256.076,Z 166.585,A -85,B 0,C 180,E1 -18575.192,E2 -18575.192} C_VEL
LIN {X 0,Y 256.043,Z 166.58,A -85,B 0,C 180,E1 -18579.145,E2 -18579.145} C_VEL
LIN {X 0,Y 256.019,Z 166.596,A -85,B 0,C 180,E1 -18583.334,E2 -18583.334} C_VEL
LIN {X 0,Y 256.03,Z 166.586,A -85,B 0,C 180,E1 -18587.827,E2 -18587.827} C_VEL
LIN {X 0,Y 256.063,Z 166.591,A -85,B 0,C 180,E1 -18590.856,E2 -18590.856} C_VEL
LIN {X 0,Y 256.121,Z 166.582,A -85,B 0,C 180,E1 -18592.865,E2 -18592.865} C_VEL
LIN {X 0,Y 256.062,Z 166.587,A -85,B 0,C 180,E1 -18596.706,E2 -18596.706} C_VEL
LIN {X 0,Y 256.049,Z 166.589,A -85,B 0,C 180,E1 -18600.392,E2 -18600.392} C_VEL
LIN {X 0,Y 256.068,Z 166.587,A -85,B 0,C 180,E1 -18603.951,E2 -18603.951} C_VEL
LIN {X 0,Y 256.051,Z 166.585,A -85,B 0,C 180,E1 -18607.401,E2 -18607.401} C_VEL
LIN {X 0,Y 256.101,Z 166.585,A -85,B 0,C 180,E1 -18610.773,E2 -18610.773} C_VEL
LIN {X 0,Y 256.206,Z 166.571,A -85,B 0,C 180,E1 -18614.079,E2 -18614.079} C_VEL
LIN {X 0,Y 256.269,Z 166.559,A -85,B 0,C 180,E1 -18618.932,E2 -18618.932} C_VEL
LIN {X 0,Y 256.429,Z 166.552,A -85,B 0,C 180,E1 -18621.263,E2 -18621.263} C_VEL
LIN {X 0,Y 256.579,Z 167.252,A -85,B 0,C 180,E1 -18621.428,E2 -18621.428} C_VEL
LIN {X 0,Y 263.268,Z 182.767,A -85,B 0,C 180,E1 -18622.671,E2 -18622.671} C_VEL
LIN {X 0,Y 269.251,Z 197.762,A -85,B 0,C 180,E1 -18623.76,E2 -18623.76} C_VEL
LIN {X 0,Y 271.189,Z 203.21,A -85,B 0,C 180,E1 -18624.118,E2 -18624.118} C_VEL
LIN {X 0,Y 269.995,Z 241.917,A -85,B 0,C 180,E1 -18625.155,E2 -18625.155} C_VEL
LIN {X 0,Y 268.8,Z 275.087,A -85,B 0,C 180,E1 -18626.083,E2 -18626.083} C_VEL
LIN {X 0,Y 267.822,Z 288.582,A -85,B 0,C 180,E1 -18626.761,E2 -18626.761} C_VEL
LIN {X 0,Y 266.793,Z 300.519,A -85,B 0,C 180,E1 -18627.66,E2 -18627.66} C_VEL
LIN {X 0,Y 265.379,Z 312.387,A -85,B 0,C 180,E1 -18628.862,E2 -18628.862} C_VEL
LIN {X 0,Y 263.624,Z 324.027,A -85,B 0,C 180,E1 -18630.382,E2 -18630.382} C_VEL
LIN {X 0,Y 261.854,Z 334.477,A -85,B 0,C 180,E1 -18632.115,E2 -18632.115} C_VEL
LIN {X 0,Y 260.255,Z 343.304,A -85,B 0,C 180,E1 -18633.943,E2 -18633.943} C_VEL
LIN {X 0,Y 258.481,Z 352.256,A -85,B 0,C 180,E1 -18636.243,E2 -18636.243} C_VEL
LIN {X 0,Y 256.946,Z 359.706,A -85,B 0,C 180,E1 -18638.652,E2 -18638.652} C_VEL
LIN {X 0,Y 255.849,Z 365.58,A -85,B 0,C 180,E1 -18641.086,E2 -18641.086} C_VEL
LIN {X 0,Y 254.972,Z 370.199,A -85,B 0,C 180,E1 -18643.55,E2 -18643.55} C_VEL
LIN {X 0,Y 254.363,Z 373.671,A -85,B 0,C 180,E1 -18646.039,E2 -18646.039} C_VEL
LIN {X 0,Y 254.038,Z 375.397,A -85,B 0,C 180,E1 -18647.717,E2 -18647.717} C_VEL
LIN {X 0,Y 253.87,Z 376.848,A -85,B 0,C 180,E1 -18649.744,E2 -18649.744} C_VEL
LIN {X 0,Y 253.803,Z 377.806,A -85,B 0,C 180,E1 -18652.809,E2 -18652.809} C_VEL
LIN {X 0,Y 253.917,Z 377.709,A -85,B 0,C 180,E1 -18654.53,E2 -18654.53} C_VEL
LIN {X 0,Y 254.121,Z 377.104,A -85,B 0,C 180,E1 -18656.263,E2 -18656.263} C_VEL
LIN {X 0,Y 254.457,Z 376.051,A -85,B 0,C 180,E1 -18658.004,E2 -18658.004} C_VEL
LIN {X 0,Y 255.193,Z 373.52,A -85,B 0,C 180,E1 -18660.621,E2 -18660.621} C_VEL
LIN {X 0,Y 256.238,Z 369.717,A -85,B 0,C 180,E1 -18663.268,E2 -18663.268} C_VEL
LIN {X 0,Y 257.715,Z 364.523,A -85,B 0,C 180,E1 -18665.896,E2 -18665.896} C_VEL
LIN {X 0,Y 259.562,Z 357.759,A -85,B 0,C 180,E1 -18668.518,E2 -18668.518} C_VEL
LIN {X 0,Y 261.45,Z 350.956,A -85,B 0,C 180,E1 -18670.591,E2 -18670.591} C_VEL
LIN {X 0,Y 263.735,Z 341.876,A -85,B 0,C 180,E1 -18672.806,E2 -18672.806} C_VEL
LIN {X 0,Y 266.122,Z 331.826,A -85,B 0,C 180,E1 -18674.739,E2 -18674.739} C_VEL
LIN {X 0,Y 268.232,Z 321.239,A -85,B 0,C 180,E1 -18676.37,E2 -18676.37} C_VEL
LIN {X 0,Y 270.235,Z 310.446,A -85,B 0,C 180,E1 -18677.654,E2 -18677.654} C_VEL
LIN {X 0,Y 271.922,Z 297.803,A -85,B 0,C 180,E1 -18678.83,E2 -18678.83} C_VEL
LIN {X 0,Y 273.218,Z 285.088,A -85,B 0,C 180,E1 -18679.68,E2 -18679.68} C_VEL
LIN {X 0,Y 274.108,Z 272.429,A -85,B 0,C 180,E1 -18680.22,E2 -18680.22} C_VEL
LIN {X 0,Y 276.694,Z 208.661,A -85,B 0,C 180,E1 -18681.917,E2 -18681.917} C_VEL
LIN {X 0,Y 270.138,Z 193.32,A -85,B 0,C 180,E1 -18683.366,E2 -18683.366} C_VEL
LIN {X 0,Y 262.773,Z 179.086,A -85,B 0,C 180,E1 -18685.017,E2 -18685.017} C_VEL
LIN {X 0,Y 258.345,Z 171.541,A -85,B 0,C 180,E1 -18686.047,E2 -18686.047} C_VEL
LIN {X 0,Y 256.482,Z 168.029,A -85,B 0,C 180,E1 -18686.55,E2 -18686.55} C_VEL
LIN {X 0,Y 256.095,Z 166.587,A -85,B 0,C 180,E1 -18687.31,E2 -18687.31} C_VEL
LIN {X 0,Y 256.136,Z 166.581,A -85,B 0,C 180,E1 -18691.406,E2 -18691.406} C_VEL
LIN {X 0,Y 256.165,Z 166.573,A -85,B 0,C 180,E1 -18695.701,E2 -18695.701} C_VEL
LIN {X 0,Y 256.165,Z 166.571,A -85,B 0,C 180,E1 -18699.106,E2 -18699.106} C_VEL
LIN {X 0,Y 256.258,Z 166.564,A -85,B 0,C 180,E1 -18704.084,E2 -18704.084} C_VEL
LIN {X 0,Y 256.28,Z 166.56,A -85,B 0,C 180,E1 -18708.687,E2 -18708.687} C_VEL
LIN {X 0,Y 256.492,Z 166.527,A -85,B 0,C 180,E1 -18712.127,E2 -18712.127} C_VEL
LIN {X 0,Y 256.332,Z 166.539,A -85,B 0,C 180,E1 -18715.486,E2 -18715.486} C_VEL
LIN {X 0,Y 255.777,Z 166.613,A -85,B 0,C 180,E1 -18716.802,E2 -18716.802} C_VEL
LIN {X 0,Y 253.121,Z 166.948,A -85,B 0,C 180,E1 -18718.953,E2 -18718.953} C_VEL
LIN {X 0,Y 249.906,Z 167.34,A -85,B 0,C 180,E1 -18721.597,E2 -18721.597} C_VEL
LIN {X 0,Y 249.489,Z 167.394,A -85,B 0,C 180,E1 -18722.511,E2 -18722.511} C_VEL
LIN {X 0,Y 249.431,Z 167.397,A -85,B 0,C 180,E1 -18726.473,E2 -18726.473} C_VEL
LIN {X 0,Y 249.344,Z 167.415,A -85,B 0,C 180,E1 -18729.738,E2 -18729.738} C_VEL
LIN {X 0,Y 249.167,Z 167.444,A -85,B 0,C 180,E1 -18734.707,E2 -18734.707} C_VEL
LIN {X 0,Y 249.094,Z 167.453,A -85,B 0,C 180,E1 -18738.082,E2 -18738.082} C_VEL
LIN {X 0,Y 249.045,Z 167.449,A -85,B 0,C 180,E1 -18741.523,E2 -18741.523} C_VEL
LIN {X 0,Y 249.05,Z 167.452,A -85,B 0,C 180,E1 -18745.443,E2 -18745.443} C_VEL
LIN {X 0,Y 249.039,Z 167.463,A -85,B 0,C 180,E1 -18748.975,E2 -18748.975} C_VEL
LIN {X 0,Y 249.03,Z 167.465,A -85,B 0,C 180,E1 -18752.427,E2 -18752.427} C_VEL
LIN {X 0,Y 249.013,Z 167.468,A -85,B 0,C 180,E1 -18756.35,E2 -18756.35} C_VEL
LIN {X 0,Y 248.974,Z 167.472,A -85,B 0,C 180,E1 -18760.486,E2 -18760.486} C_VEL
LIN {X 0,Y 248.965,Z 167.477,A -85,B 0,C 180,E1 -18764.889,E2 -18764.889} C_VEL
LIN {X 0,Y 248.971,Z 167.489,A -85,B 0,C 180,E1 -18768.259,E2 -18768.259} C_VEL
LIN {X 0,Y 251.591,Z 176.577,A -85,B 0,C 180,E1 -18772.587,E2 -18772.587} C_VEL
LIN {X 0,Y 252.933,Z 181.84,A -85,B 0,C 180,E1 -18774.88,E2 -18774.88} C_VEL
LIN {X 0,Y 255.141,Z 186.214,A -85,B 0,C 180,E1 -18775.446,E2 -18775.446} C_VEL
LIN {X 0,Y 261.676,Z 199.646,A -85,B 0,C 180,E1 -18777.05,E2 -18777.05} C_VEL
LIN {X 0,Y 266.101,Z 210.283,A -85,B 0,C 180,E1 -18778.115,E2 -18778.115} C_VEL
LIN {X 0,Y 269.424,Z 232.784,A -85,B 0,C 180,E1 -18779.363,E2 -18779.363} C_VEL
LIN {X 0,Y 269.726,Z 236.527,A -85,B 0,C 180,E1 -18779.53,E2 -18779.53} C_VEL
LIN {X 0,Y 267.542,Z 291.572,A -85,B 0,C 180,E1 -18781.074,E2 -18781.074} C_VEL
LIN {X 0,Y 266.167,Z 305.389,A -85,B 0,C 180,E1 -18781.73,E2 -18781.73} C_VEL
LIN {X 0,Y 264.426,Z 317.722,A -85,B 0,C 180,E1 -18782.604,E2 -18782.604} C_VEL
LIN {X 0,Y 262.364,Z 329.575,A -85,B 0,C 180,E1 -18783.769,E2 -18783.769} C_VEL
LIN {X 0,Y 260.027,Z 340.985,A -85,B 0,C 180,E1 -18785.233,E2 -18785.233} C_VEL
LIN {X 0,Y 257.612,Z 351.308,A -85,B 0,C 180,E1 -18786.911,E2 -18786.911} C_VEL
LIN {X 0,Y 255.431,Z 359.773,A -85,B 0,C 180,E1 -18788.619,E2 -18788.619} C_VEL
LIN {X 0,Y 253.249,Z 368.6,A -85,B 0,C 180,E1 -18790.855,E2 -18790.855} C_VEL
LIN {X 0,Y 251.139,Z 376.402,A -85,B 0,C 180,E1 -18793.331,E2 -18793.331} C_VEL
LIN {X 0,Y 249.154,Z 383.273,A -85,B 0,C 180,E1 -18796.128,E2 -18796.128} C_VEL
LIN {X 0,Y 248.091,Z 387.829,A -85,B 0,C 180,E1 -18798.563,E2 -18798.563} C_VEL
LIN {X 0,Y 247.591,Z 390.244,A -85,B 0,C 180,E1 -18800.194,E2 -18800.194} C_VEL
LIN {X 0,Y 247.208,Z 392.234,A -85,B 0,C 180,E1 -18801.828,E2 -18801.828} C_VEL
LIN {X 0,Y 246.982,Z 393.811,A -85,B 0,C 180,E1 -18803.465,E2 -18803.465} C_VEL
LIN {X 0,Y 246.886,Z 394.94,A -85,B 0,C 180,E1 -18805.101,E2 -18805.101} C_VEL
LIN {X 0,Y 246.898,Z 395.667,A -85,B 0,C 180,E1 -18806.737,E2 -18806.737} C_VEL
LIN {X 0,Y 246.978,Z 396.008,A -85,B 0,C 180,E1 -18808.37,E2 -18808.37} C_VEL
LIN {X 0,Y 247.03,Z 395.955,A -85,B 0,C 180,E1 -18810,E2 -18810} C_VEL
LIN {X 0,Y 247.007,Z 395.463,A -85,B 0,C 180,E1 -18811.631,E2 -18811.631} C_VEL
LIN {X 0,Y 246.916,Z 394.554,A -85,B 0,C 180,E1 -18813.264,E2 -18813.264} C_VEL
LIN {X 0,Y 246.886,Z 393.242,A -85,B 0,C 180,E1 -18814.899,E2 -18814.899} C_VEL
LIN {X 0,Y 247.1,Z 390.449,A -85,B 0,C 180,E1 -18817.354,E2 -18817.354} C_VEL
LIN {X 0,Y 247.54,Z 386.607,A -85,B 0,C 180,E1 -18819.808,E2 -18819.808} C_VEL
LIN {X 0,Y 248.258,Z 381.615,A -85,B 0,C 180,E1 -18822.259,E2 -18822.259} C_VEL
LIN {X 0,Y 249.474,Z 375.334,A -85,B 0,C 180,E1 -18824.688,E2 -18824.688} C_VEL
LIN {X 0,Y 251.088,Z 367.468,A -85,B 0,C 180,E1 -18827.092,E2 -18827.092} C_VEL
LIN {X 0,Y 252.688,Z 358.611,A -85,B 0,C 180,E1 -18829.262,E2 -18829.262} C_VEL
LIN {X 0,Y 254.552,Z 348.496,A -85,B 0,C 180,E1 -18831.246,E2 -18831.246} C_VEL
LIN {X 0,Y 256.669,Z 337.228,A -85,B 0,C 180,E1 -18832.967,E2 -18832.967} C_VEL
LIN {X 0,Y 258.454,Z 326.186,A -85,B 0,C 180,E1 -18834.286,E2 -18834.286} C_VEL
LIN {X 0,Y 260.095,Z 313.974,A -85,B 0,C 180,E1 -18835.402,E2 -18835.402} C_VEL
LIN {X 0,Y 261.355,Z 301.216,A -85,B 0,C 180,E1 -18836.233,E2 -18836.233} C_VEL
LIN {X 0,Y 262.205,Z 287.894,A -85,B 0,C 180,E1 -18836.785,E2 -18836.785} C_VEL
LIN {X 0,Y 263.903,Z 233.307,A -85,B 0,C 180,E1 -18838.297,E2 -18838.297} C_VEL
LIN {X 0,Y 259.359,Z 201.162,A -85,B 0,C 180,E1 -18839.774,E2 -18839.774} C_VEL
LIN {X 0,Y 253.82,Z 186.54,A -85,B 0,C 180,E1 -18840.865,E2 -18840.865} C_VEL
LIN {X 0,Y 252.604,Z 183.347,A -85,B 0,C 180,E1 -18841.131,E2 -18841.131} C_VEL
LIN {X 0,Y 250.563,Z 173.814,A -85,B 0,C 180,E1 -18844.749,E2 -18844.749} C_VEL
LIN {X 0,Y 249.059,Z 167.463,A -85,B 0,C 180,E1 -18847.345,E2 -18847.345} C_VEL
LIN {X 0,Y 248.976,Z 167.474,A -85,B 0,C 180,E1 -18850.485,E2 -18850.485} C_VEL
LIN {X 0,Y 248.967,Z 167.473,A -85,B 0,C 180,E1 -18854.888,E2 -18854.888} C_VEL
LIN {X 0,Y 248.984,Z 167.473,A -85,B 0,C 180,E1 -18857.355,E2 -18857.355} C_VEL
LIN {X 0,Y 249.046,Z 167.463,A -85,B 0,C 180,E1 -18862.201,E2 -18862.201} C_VEL
LIN {X 0,Y 249.048,Z 167.463,A -85,B 0,C 180,E1 -18865.639,E2 -18865.639} C_VEL
LIN {X 0,Y 249.007,Z 167.468,A -85,B 0,C 180,E1 -18869.466,E2 -18869.466} C_VEL
LIN {X 0,Y 249.04,Z 167.465,A -85,B 0,C 180,E1 -18873.157,E2 -18873.157} C_VEL
LIN {X 0,Y 249.056,Z 167.463,A -85,B 0,C 180,E1 -18876.729,E2 -18876.729} C_VEL
LIN {X 0,Y 249.049,Z 167.461,A -85,B 0,C 180,E1 -18880.205,E2 -18880.205} C_VEL
LIN {X 0,Y 249.162,Z 167.447,A -85,B 0,C 180,E1 -18883.615,E2 -18883.615} C_VEL
LIN {X 0,Y 249.234,Z 167.436,A -85,B 0,C 180,E1 -18888.614,E2 -18888.614} C_VEL
LIN {X 0,Y 249.422,Z 167.399,A -85,B 0,C 180,E1 -18891.9,E2 -18891.9} C_VEL
